LIN {X 0,Y 337.029,Z 979.559,A -85,B 0,C 180,E1 7222.353,E2 7222.353} C_VEL
LIN {X 0,Y 341.956,Z 956.533,A -85,B 0,C 180,E1 7221.821,E2 7221.821} C_VEL
LIN {X 0,Y 345.106,Z 934.145,A -85,B 0,C 180,E1 7221.412,E2 7221.412} C_VEL
LIN {X 0,Y 361.472,Z 765.013,A -85,B 0,C 180,E1 7218.829,E2 7218.829} C_VEL
LIN {X 0,Y 358.291,Z 755.839,A -85,B 0,C 180,E1 7216.122,E2 7216.122} C_VEL
LIN {X 0,Y 355.543,Z 748.18,A -85,B 0,C 180,E1 7213.167,E2 7213.167} C_VEL
LIN {X 0,Y 353.615,Z 742.614,A -85,B 0,C 180,E1 7210.344,E2 7210.344} C_VEL
LIN {X 0,Y 352.385,Z 739.021,A -85,B 0,C 180,E1 7207.664,E2 7207.664} C_VEL
LIN {X 0,Y 351.824,Z 736.43,A -85,B 0,C 180,E1 7205.055,E2 7205.055} C_VEL
LIN {X 0,Y 352.166,Z 735.346,A -85,B 0,C 180,E1 7200.651,E2 7200.651} C_VEL
LIN {X 0,Y 353.212,Z 736.345,A -85,B 0,C 180,E1 7197.891,E2 7197.891} C_VEL
LIN {X 0,Y 354.815,Z 738.293,A -85,B 0,C 180,E1 7195.312,E2 7195.312} C_VEL
LIN {X 0,Y 357.247,Z 742.275,A -85,B 0,C 180,E1 7192.441,E2 7192.441} C_VEL
LIN {X 0,Y 359.812,Z 746.722,A -85,B 0,C 180,E1 7190.079,E2 7190.079} C_VEL
LIN {X 0,Y 363.341,Z 753.377,A -85,B 0,C 180,E1 7187.385,E2 7187.385} C_VEL
LIN {X 0,Y 361.606,Z 770.162,A -85,B 0,C 180,E1 7187.124,E2 7187.124} C_VEL
LIN {X 0,Y 360.533,Z 777.852,A -85,B 0,C 180,E1 7187.159,E2 7187.159} C_VEL
LIN {X 0,Y 356.723,Z 798.361,A -85,B 0,C 180,E1 7187.805,E2 7187.805} C_VEL
LIN {X 0,Y 355.838,Z 804.96,A -85,B 0,C 180,E1 7187.82,E2 7187.82} C_VEL
LIN {X 0,Y 342.283,Z 933.926,A -85,B 0,C 180,E1 7185.77,E2 7185.77} C_VEL
LIN {X 0,Y 338.154,Z 957.934,A -85,B 0,C 180,E1 7185.264,E2 7185.264} C_VEL
LIN {X 0,Y 333.158,Z 979.434,A -85,B 0,C 180,E1 7184.668,E2 7184.668} C_VEL
LIN {X 0,Y 326.772,Z 1000.882,A -85,B 0,C 180,E1 7183.899,E2 7183.899} C_VEL
LIN {X 0,Y 319.517,Z 1021.265,A -85,B 0,C 180,E1 7182.976,E2 7182.976} C_VEL
LIN {X 0,Y 310.546,Z 1042.479,A -85,B 0,C 180,E1 7181.769,E2 7181.769} C_VEL
LIN {X 0,Y 300.999,Z 1062.082,A -85,B 0,C 180,E1 7180.396,E2 7180.396} C_VEL
LIN {X 0,Y 289.845,Z 1081.992,A -85,B 0,C 180,E1 7178.654,E2 7178.654} C_VEL
LIN {X 0,Y 278.251,Z 1100.526,A -85,B 0,C 180,E1 7176.65,E2 7176.65} C_VEL
LIN {X 0,Y 266.028,Z 1117.83,A -85,B 0,C 180,E1 7174.289,E2 7174.289} C_VEL
LIN {X 0,Y 253.22,Z 1134.476,A -85,B 0,C 180,E1 7171.459,E2 7171.459} C_VEL
LIN {X 0,Y 240.898,Z 1149.035,A -85,B 0,C 180,E1 7168.305,E2 7168.305} C_VEL
LIN {X 0,Y 227.747,Z 1163.57,A -85,B 0,C 180,E1 7164.31,E2 7164.31} C_VEL
LIN {X 0,Y 216.336,Z 1175.4,A -85,B 0,C 180,E1 7160.104,E2 7160.104} C_VEL
LIN {X 0,Y 204.152,Z 1187.573,A -85,B 0,C 180,E1 7154.456,E2 7154.456} C_VEL
LIN {X 0,Y 194.783,Z 1196.854,A -85,B 0,C 180,E1 7148.774,E2 7148.774} C_VEL
LIN {X 0,Y 186.937,Z 1204.75,A -85,B 0,C 180,E1 7142.316,E2 7142.316} C_VEL
LIN {X 0,Y 181.505,Z 1210.761,A -85,B 0,C 180,E1 7135.797,E2 7135.797} C_VEL
LIN {X 0,Y 177.788,Z 1215.641,A -85,B 0,C 180,E1 7128.357,E2 7128.357} C_VEL
LIN {X 0,Y 176.331,Z 1218.412,A -85,B 0,C 180,E1 7122.111,E2 7122.111} C_VEL
LIN {X 0,Y 175.975,Z 1220.093,A -85,B 0,C 180,E1 7115.87,E2 7115.87} C_VEL
LIN {X 0,Y 176.025,Z 1220.645,A -85,B 0,C 180,E1 7110,E2 7110} C_VEL
LIN {X 0,Y 175.975,Z 1220.076,A -85,B 0,C 180,E1 7104.13,E2 7104.13} C_VEL
LIN {X 0,Y 176.331,Z 1218.382,A -85,B 0,C 180,E1 7097.889,E2 7097.889} C_VEL
LIN {X 0,Y 177.901,Z 1215.431,A -85,B 0,C 180,E1 7091.315,E2 7091.315} C_VEL
LIN {X 0,Y 181.934,Z 1210.166,A -85,B 0,C 180,E1 7083.567,E2 7083.567} C_VEL
LIN {X 0,Y 187.569,Z 1204.025,A -85,B 0,C 180,E1 7077.063,E2 7077.063} C_VEL
LIN {X 0,Y 195.996,Z 1195.489,A -85,B 0,C 180,E1 7070.381,E2 7070.381} C_VEL
LIN {X 0,Y 205.627,Z 1186.035,A -85,B 0,C 180,E1 7064.772,E2 7064.772} C_VEL
LIN {X 0,Y 216.893,Z 1174.659,A -85,B 0,C 180,E1 7059.659,E2 7059.659} C_VEL
LIN {X 0,Y 229.005,Z 1162.095,A -85,B 0,C 180,E1 7055.268,E2 7055.268} C_VEL
LIN {X 0,Y 241.566,Z 1148.034,A -85,B 0,C 180,E1 7051.499,E2 7051.499} C_VEL
LIN {X 0,Y 254.307,Z 1132.865,A -85,B 0,C 180,E1 7048.273,E2 7048.273} C_VEL
LIN {X 0,Y 266.218,Z 1117.253,A -85,B 0,C 180,E1 7045.659,E2 7045.659} C_VEL
LIN {X 0,Y 278.624,Z 1099.559,A -85,B 0,C 180,E1 7043.268,E2 7043.268} C_VEL
LIN {X 0,Y 289.825,Z 1081.596,A -85,B 0,C 180,E1 7041.336,E2 7041.336} C_VEL
LIN {X 0,Y 300.817,Z 1061.918,A -85,B 0,C 180,E1 7039.616,E2 7039.616} C_VEL
LIN {X 0,Y 310.102,Z 1042.861,A -85,B 0,C 180,E1 7038.277,E2 7038.277} C_VEL
LIN {X 0,Y 319.595,Z 1020.331,A -85,B 0,C 180,E1 7036.999,E2 7036.999} C_VEL
LIN {X 0,Y 327.182,Z 998.816,A -85,B 0,C 180,E1 7036.034,E2 7036.034} C_VEL
LIN {X 0,Y 333.952,Z 975.076,A -85,B 0,C 180,E1 7035.212,E2 7035.212} C_VEL
LIN {X 0,Y 339.074,Z 952.161,A -85,B 0,C 180,E1 7034.611,E2 7034.611} C_VEL
LIN {X 0,Y 342.693,Z 928.355,A -85,B 0,C 180,E1 7034.15,E2 7034.15} C_VEL
LIN {X 0,Y 360.379,Z 758.499,A -85,B 0,C 180,E1 7031.465,E2 7031.465} C_VEL
LIN {X 0,Y 356.925,Z 751.817,A -85,B 0,C 180,E1 7028.539,E2 7028.539} C_VEL
LIN {X 0,Y 354.566,Z 747.889,A -85,B 0,C 180,E1 7026.07,E2 7026.07} C_VEL
LIN {X 0,Y 352.955,Z 745.226,A -85,B 0,C 180,E1 7023.899,E2 7023.899} C_VEL
LIN {X 0,Y 351.105,Z 743.014,A -85,B 0,C 180,E1 7020.163,E2 7020.163} C_VEL
LIN {X 0,Y 350.436,Z 743.287,A -85,B 0,C 180,E1 7016.892,E2 7016.892} C_VEL
LIN {X 0,Y 350.601,Z 744.712,A -85,B 0,C 180,E1 7014.107,E2 7014.107} C_VEL
LIN {X 0,Y 351.499,Z 748.289,A -85,B 0,C 180,E1 7011.081,E2 7011.081} C_VEL
LIN {X 0,Y 352.83,Z 752.197,A -85,B 0,C 180,E1 7008.641,E2 7008.641} C_VEL
LIN {X 0,Y 355.185,Z 759.277,A -85,B 0,C 180,E1 7005.565,E2 7005.565} C_VEL
LIN {X 0,Y 357.437,Z 765.972,A -85,B 0,C 180,E1 7003.296,E2 7003.296} C_VEL
LIN {X 0,Y 358.652,Z 769.729,A -85,B 0,C 180,E1 7002.216,E2 7002.216} C_VEL
LIN {X 0,Y 341.49,Z 941.423,A -85,B 0,C 180,E1 6999.633,E2 6999.633} C_VEL
LIN {X 0,Y 337.472,Z 964.923,A -85,B 0,C 180,E1 6999.174,E2 6999.174} C_VEL
LIN {X 0,Y 332.156,Z 987.28,A -85,B 0,C 180,E1 6998.628,E2 6998.628} C_VEL
LIN {X 0,Y 325.487,Z 1008.737,A -85,B 0,C 180,E1 6997.92,E2 6997.92} C_VEL
LIN {X 0,Y 317.241,Z 1030.712,A -85,B 0,C 180,E1 6996.971,E2 6996.971} C_VEL
LIN {X 0,Y 308.826,Z 1049.617,A -85,B 0,C 180,E1 6995.924,E2 6995.924} C_VEL
LIN {X 0,Y 298.079,Z 1070.431,A -85,B 0,C 180,E1 6994.464,E2 6994.464} C_VEL
LIN {X 0,Y 287.177,Z 1088.966,A -85,B 0,C 180,E1 6992.819,E2 6992.819} C_VEL
LIN {X 0,Y 275.368,Z 1106.536,A -85,B 0,C 180,E1 6990.838,E2 6990.838} C_VEL
LIN {X 0,Y 263.584,Z 1122.475,A -85,B 0,C 180,E1 6988.594,E2 6988.594} C_VEL
LIN {X 0,Y 250.684,Z 1138.039,A -85,B 0,C 180,E1 6985.778,E2 6985.778} C_VEL
LIN {X 0,Y 237.366,Z 1152.752,A -85,B 0,C 180,E1 6982.352,E2 6982.352} C_VEL
LIN {X 0,Y 225.05,Z 1165.313,A -85,B 0,C 180,E1 6978.547,E2 6978.547} C_VEL
LIN {X 0,Y 213.031,Z 1176.669,A -85,B 0,C 180,E1 6973.998,E2 6973.998} C_VEL
LIN {X 0,Y 202.334,Z 1186.397,A -85,B 0,C 180,E1 6968.872,E2 6968.872} C_VEL
LIN {X 0,Y 193.318,Z 1194.256,A -85,B 0,C 180,E1 6963.246,E2 6963.246} C_VEL
LIN {X 0,Y 185.318,Z 1201.367,A -85,B 0,C 180,E1 6956.258,E2 6956.258} C_VEL
LIN {X 0,Y 180.263,Z 1206.2,A -85,B 0,C 180,E1 6949.439,E2 6949.439} C_VEL
LIN {X 0,Y 177.256,Z 1209.525,A -85,B 0,C 180,E1 6942.047,E2 6942.047} C_VEL
LIN {X 0,Y 176.192,Z 1211.235,A -85,B 0,C 180,E1 6935.209,E2 6935.209} C_VEL
LIN {X 0,Y 176.053,Z 1211.594,A -85,B 0,C 180,E1 6929.024,E2 6929.024} C_VEL
LIN {X 0,Y 176.351,Z 1210.882,A -85,B 0,C 180,E1 6922.835,E2 6922.835} C_VEL
LIN {X 0,Y 177.913,Z 1208.822,A -85,B 0,C 180,E1 6915.684,E2 6915.684} C_VEL
LIN {X 0,Y 181.579,Z 1204.916,A -85,B 0,C 180,E1 6908.35,E2 6908.35} C_VEL
LIN {X 0,Y 187.946,Z 1199.095,A -85,B 0,C 180,E1 6901.046,E2 6901.046} C_VEL
LIN {X 0,Y 195.617,Z 1192.379,A -85,B 0,C 180,E1 6895.078,E2 6895.078} C_VEL
LIN {X 0,Y 205.605,Z 1183.544,A -85,B 0,C 180,E1 6889.335,E2 6889.335} C_VEL
LIN {X 0,Y 216.822,Z 1173.386,A -85,B 0,C 180,E1 6884.376,E2 6884.376} C_VEL
LIN {X 0,Y 228.831,Z 1161.702,A -85,B 0,C 180,E1 6880.125,E2 6880.125} C_VEL
LIN {X 0,Y 241.968,Z 1148.06,A -85,B 0,C 180,E1 6876.315,E2 6876.315} C_VEL
LIN {X 0,Y 253.902,Z 1134.56,A -85,B 0,C 180,E1 6873.4,E2 6873.4} C_VEL
LIN {X 0,Y 267.191,Z 1118.005,A -85,B 0,C 180,E1 6870.607,E2 6870.607} C_VEL
LIN {X 0,Y 279.516,Z 1101.047,A -85,B 0,C 180,E1 6868.362,E2 6868.362} C_VEL
LIN {X 0,Y 291.037,Z 1083.022,A -85,B 0,C 180,E1 6866.498,E2 6866.498} C_VEL
LIN {X 0,Y 302.045,Z 1063.664,A -85,B 0,C 180,E1 6864.904,E2 6864.904} C_VEL
LIN {X 0,Y 311.514,Z 1044.454,A -85,B 0,C 180,E1 6863.655,E2 6863.655} C_VEL
LIN {X 0,Y 320.499,Z 1023.203,A -85,B 0,C 180,E1 6862.565,E2 6862.565} C_VEL
LIN {X 0,Y 327.791,Z 1002.724,A -85,B 0,C 180,E1 6861.75,E2 6861.75} C_VEL
LIN {X 0,Y 334.252,Z 980.148,A -85,B 0,C 180,E1 6861.076,E2 6861.076} C_VEL
LIN {X 0,Y 339.282,Z 957.394,A -85,B 0,C 180,E1 6860.559,E2 6860.559} C_VEL
LIN {X 0,Y 342.592,Z 934.57,A -85,B 0,C 180,E1 6860.148,E2 6860.148} C_VEL
LIN {X 0,Y 358.93,Z 769.805,A -85,B 0,C 180,E1 6857.677,E2 6857.677} C_VEL
LIN {X 0,Y 355.989,Z 761.006,A -85,B 0,C 180,E1 6854.892,E2 6854.892} C_VEL
LIN {X 0,Y 353.97,Z 755.084,A -85,B 0,C 180,E1 6852.48,E2 6852.48} C_VEL
LIN {X 0,Y 352.395,Z 750.208,A -85,B 0,C 180,E1 6849.967,E2 6849.967} C_VEL
LIN {X 0,Y 351.295,Z 746.748,A -85,B 0,C 180,E1 6847.359,E2 6847.359} C_VEL
LIN {X 0,Y 350.827,Z 744.326,A -85,B 0,C 180,E1 6844.905,E2 6844.905} C_VEL
LIN {X 0,Y 351.177,Z 743.286,A -85,B 0,C 180,E1 6840.653,E2 6840.653} C_VEL
LIN {X 0,Y 352.164,Z 744.248,A -85,B 0,C 180,E1 6837.999,E2 6837.999} C_VEL
LIN {X 0,Y 353.698,Z 746.195,A -85,B 0,C 180,E1 6835.46,E2 6835.46} C_VEL
LIN {X 0,Y 356.004,Z 750.089,A -85,B 0,C 180,E1 6832.658,E2 6832.658} C_VEL
LIN {X 0,Y 358.693,Z 754.882,A -85,B 0,C 180,E1 6830.129,E2 6830.129} C_VEL
LIN {X 0,Y 360.649,Z 758.948,A -85,B 0,C 180,E1 6828.524,E2 6828.524} C_VEL
LIN {X 0,Y 355.838,Z 804.96,A -85,B 0,C 180,E1 6827.82,E2 6827.82} C_VEL
LIN {X 0,Y 354.777,Z 812.65,A -85,B 0,C 180,E1 6827.857,E2 6827.857} C_VEL
LIN {X 0,Y 351.023,Z 833.156,A -85,B 0,C 180,E1 6828.524,E2 6828.524} C_VEL
LIN {X 0,Y 350.133,Z 839.755,A -85,B 0,C 180,E1 6828.543,E2 6828.543} C_VEL
LIN {X 0,Y 339.9,Z 934.846,A -85,B 0,C 180,E1 6827.045,E2 6827.045} C_VEL
LIN {X 0,Y 335.705,Z 958.6,A -85,B 0,C 180,E1 6826.554,E2 6826.554} C_VEL
LIN {X 0,Y 330.459,Z 980.726,A -85,B 0,C 180,E1 6825.954,E2 6825.954} C_VEL
LIN {X 0,Y 323.727,Z 1002.609,A -85,B 0,C 180,E1 6825.178,E2 6825.178} C_VEL
LIN {X 0,Y 315.704,Z 1024.466,A -85,B 0,C 180,E1 6824.194,E2 6824.194} C_VEL
LIN {X 0,Y 306.366,Z 1045.56,A -85,B 0,C 180,E1 6822.986,E2 6822.986} C_VEL
LIN {X 0,Y 295.733,Z 1066.415,A -85,B 0,C 180,E1 6821.506,E2 6821.506} C_VEL
LIN {X 0,Y 285.197,Z 1084.461,A -85,B 0,C 180,E1 6819.905,E2 6819.905} C_VEL
LIN {X 0,Y 272.268,Z 1104.152,A -85,B 0,C 180,E1 6817.733,E2 6817.733} C_VEL
LIN {X 0,Y 260.434,Z 1120.317,A -85,B 0,C 180,E1 6815.49,E2 6815.49} C_VEL
LIN {X 0,Y 246.783,Z 1137.196,A -85,B 0,C 180,E1 6812.535,E2 6812.535} C_VEL
LIN {X 0,Y 233.842,Z 1151.914,A -85,B 0,C 180,E1 6809.253,E2 6809.253} C_VEL
LIN {X 0,Y 220.408,Z 1165.925,A -85,B 0,C 180,E1 6805.194,E2 6805.194} C_VEL
LIN {X 0,Y 208.173,Z 1178.082,A -85,B 0,C 180,E1 6800.649,E2 6800.649} C_VEL
LIN {X 0,Y 196.781,Z 1188.765,A -85,B 0,C 180,E1 6795.345,E2 6795.345} C_VEL
LIN {X 0,Y 186.709,Z 1198.208,A -85,B 0,C 180,E1 6789.191,E2 6789.191} C_VEL
LIN {X 0,Y 178.738,Z 1205.78,A -85,B 0,C 180,E1 6782.481,E2 6782.481} C_VEL
LIN {X 0,Y 172.554,Z 1212.286,A -85,B 0,C 180,E1 6774.527,E2 6774.527} C_VEL
LIN {X 0,Y 169.474,Z 1216.272,A -85,B 0,C 180,E1 6767.511,E2 6767.511} C_VEL
LIN {X 0,Y 168.095,Z 1219.159,A -85,B 0,C 180,E1 6759.587,E2 6759.587} C_VEL
LIN {X 0,Y 167.988,Z 1220.21,A -85,B 0,C 180,E1 6753.412,E2 6753.412} C_VEL
LIN {X 0,Y 168.009,Z 1220.326,A -85,B 0,C 180,E1 6748.295,E2 6748.295} C_VEL
LIN {X 0,Y 167.997,Z 1219.652,A -85,B 0,C 180,E1 6742.82,E2 6742.82} C_VEL
LIN {X 0,Y 168.51,Z 1217.933,A -85,B 0,C 180,E1 6736.62,E2 6736.62} C_VEL
LIN {X 0,Y 170.726,Z 1214.534,A -85,B 0,C 180,E1 6729.069,E2 6729.069} C_VEL
LIN {X 0,Y 175.265,Z 1209.229,A -85,B 0,C 180,E1 6721.471,E2 6721.471} C_VEL
LIN {X 0,Y 182.19,Z 1202.401,A -85,B 0,C 180,E1 6714.317,E2 6714.317} C_VEL
LIN {X 0,Y 191.024,Z 1194.007,A -85,B 0,C 180,E1 6707.935,E2 6707.935} C_VEL
LIN {X 0,Y 201.99,Z 1183.772,A -85,B 0,C 180,E1 6702.055,E2 6702.055} C_VEL
LIN {X 0,Y 212.898,Z 1173.24,A -85,B 0,C 180,E1 6697.468,E2 6697.468} C_VEL
LIN {X 0,Y 226.306,Z 1159.694,A -85,B 0,C 180,E1 6692.918,E2 6692.918} C_VEL
LIN {X 0,Y 238.766,Z 1146.183,A -85,B 0,C 180,E1 6689.423,E2 6689.423} C_VEL
LIN {X 0,Y 252.747,Z 1129.72,A -85,B 0,C 180,E1 6686.104,E2 6686.104} C_VEL
LIN {X 0,Y 265.241,Z 1113.644,A -85,B 0,C 180,E1 6683.553,E2 6683.553} C_VEL
LIN {X 0,Y 277.898,Z 1095.46,A -85,B 0,C 180,E1 6681.273,E2 6681.273} C_VEL
LIN {X 0,Y 289.428,Z 1077.105,A -85,B 0,C 180,E1 6679.421,E2 6679.421} C_VEL
LIN {X 0,Y 300.367,Z 1057.12,A -85,B 0,C 180,E1 6677.819,E2 6677.819} C_VEL
LIN {X 0,Y 310.441,Z 1036.194,A -85,B 0,C 180,E1 6676.465,E2 6676.465} C_VEL
LIN {X 0,Y 318.459,Z 1016.545,A -85,B 0,C 180,E1 6675.447,E2 6675.447} C_VEL
LIN {X 0,Y 326.104,Z 994.574,A -85,B 0,C 180,E1 6674.527,E2 6674.527} C_VEL
LIN {X 0,Y 332.333,Z 972.111,A -85,B 0,C 180,E1 6673.804,E2 6673.804} C_VEL
LIN {X 0,Y 337.707,Z 946.629,A -85,B 0,C 180,E1 6673.192,E2 6673.192} C_VEL
LIN {X 0,Y 341.067,Z 923.287,A -85,B 0,C 180,E1 6672.775,E2 6672.775} C_VEL
LIN {X 0,Y 357.834,Z 764.018,A -85,B 0,C 180,E1 6670.302,E2 6670.302} C_VEL
LIN {X 0,Y 354.927,Z 758.432,A -85,B 0,C 180,E1 6667.609,E2 6667.609} C_VEL
LIN {X 0,Y 353.161,Z 755.368,A -85,B 0,C 180,E1 6665.606,E2 6665.606} C_VEL
LIN {X 0,Y 351.853,Z 753.098,A -85,B 0,C 180,E1 6663.748,E2 6663.748} C_VEL
LIN {X 0,Y 350.116,Z 750.958,A -85,B 0,C 180,E1 6660.164,E2 6660.164} C_VEL
LIN {X 0,Y 349.463,Z 751.211,A -85,B 0,C 180,E1 6656.982,E2 6656.982} C_VEL
LIN {X 0,Y 349.579,Z 752.427,A -85,B 0,C 180,E1 6654.419,E2 6654.419} C_VEL
LIN {X 0,Y 350.452,Z 756.238,A -85,B 0,C 180,E1 6651.22,E2 6651.22} C_VEL
LIN {X 0,Y 351.633,Z 759.943,A -85,B 0,C 180,E1 6648.934,E2 6648.934} C_VEL
LIN {X 0,Y 353.806,Z 766.851,A -85,B 0,C 180,E1 6645.934,E2 6645.934} C_VEL
LIN {X 0,Y 355.94,Z 773.524,A -85,B 0,C 180,E1 6643.685,E2 6643.685} C_VEL
LIN {X 0,Y 356.225,Z 774.674,A -85,B 0,C 180,E1 6643.392,E2 6643.392} C_VEL
LIN {X 0,Y 339.205,Z 941.139,A -85,B 0,C 180,E1 6640.929,E2 6640.929} C_VEL
LIN {X 0,Y 335.127,Z 964.63,A -85,B 0,C 180,E1 6640.482,E2 6640.482} C_VEL
LIN {X 0,Y 329.687,Z 987.161,A -85,B 0,C 180,E1 6639.95,E2 6639.95} C_VEL
LIN {X 0,Y 323.312,Z 1007.456,A -85,B 0,C 180,E1 6639.308,E2 6639.308} C_VEL
LIN {X 0,Y 315.069,Z 1029.359,A -85,B 0,C 180,E1 6638.407,E2 6638.407} C_VEL
LIN {X 0,Y 306.079,Z 1049.291,A -85,B 0,C 180,E1 6637.343,E2 6637.343} C_VEL
LIN {X 0,Y 295.167,Z 1070.096,A -85,B 0,C 180,E1 6635.93,E2 6635.93} C_VEL
LIN {X 0,Y 284.01,Z 1088.714,A -85,B 0,C 180,E1 6634.322,E2 6634.322} C_VEL
LIN {X 0,Y 271.939,Z 1106.33,A -85,B 0,C 180,E1 6632.387,E2 6632.387} C_VEL
LIN {X 0,Y 259.478,Z 1122.768,A -85,B 0,C 180,E1 6630.112,E2 6630.112} C_VEL
LIN {X 0,Y 246.74,Z 1137.745,A -85,B 0,C 180,E1 6627.445,E2 6627.445} C_VEL
LIN {X 0,Y 233.226,Z 1152.292,A -85,B 0,C 180,E1 6624.121,E2 6624.121} C_VEL
LIN {X 0,Y 221.236,Z 1164.119,A -85,B 0,C 180,E1 6620.608,E2 6620.608} C_VEL
LIN {X 0,Y 208.421,Z 1175.889,A -85,B 0,C 180,E1 6616.021,E2 6616.021} C_VEL
LIN {X 0,Y 197.073,Z 1185.776,A -85,B 0,C 180,E1 6610.881,E2 6610.881} C_VEL
LIN {X 0,Y 186.99,Z 1194.129,A -85,B 0,C 180,E1 6604.9,E2 6604.9} C_VEL
LIN {X 0,Y 178.69,Z 1201.085,A -85,B 0,C 180,E1 6598.036,E2 6598.036} C_VEL
LIN {X 0,Y 173.051,Z 1206.011,A -85,B 0,C 180,E1 6590.991,E2 6590.991} C_VEL
LIN {X 0,Y 169.48,Z 1209.623,A -85,B 0,C 180,E1 6582.955,E2 6582.955} C_VEL
LIN {X 0,Y 168.261,Z 1211.31,A -85,B 0,C 180,E1 6576.14,E2 6576.14} C_VEL
LIN {X 0,Y 168.054,Z 1211.842,A -85,B 0,C 180,E1 6569.659,E2 6569.659} C_VEL
LIN {X 0,Y 168.315,Z 1211.216,A -85,B 0,C 180,E1 6563.177,E2 6563.177} C_VEL
LIN {X 0,Y 169.652,Z 1209.467,A -85,B 0,C 180,E1 6556.365,E2 6556.365} C_VEL
LIN {X 0,Y 173.416,Z 1205.721,A -85,B 0,C 180,E1 6548.346,E2 6548.346} C_VEL
LIN {X 0,Y 179.567,Z 1200.472,A -85,B 0,C 180,E1 6541.025,E2 6541.025} C_VEL
LIN {X 0,Y 187.732,Z 1193.622,A -85,B 0,C 180,E1 6534.512,E2 6534.512} C_VEL
LIN {X 0,Y 197.975,Z 1185.108,A -85,B 0,C 180,E1 6528.578,E2 6528.578} C_VEL
LIN {X 0,Y 208.881,Z 1175.638,A -85,B 0,C 180,E1 6523.714,E2 6523.714} C_VEL
LIN {X 0,Y 221.785,Z 1163.78,A -85,B 0,C 180,E1 6519.137,E2 6519.137} C_VEL
LIN {X 0,Y 234.717,Z 1151.027,A -85,B 0,C 180,E1 6515.406,E2 6515.406} C_VEL
LIN {X 0,Y 248.074,Z 1136.498,A -85,B 0,C 180,E1 6512.178,E2 6512.178} C_VEL
LIN {X 0,Y 261.258,Z 1120.816,A -85,B 0,C 180,E1 6509.464,E2 6509.464} C_VEL
LIN {X 0,Y 273.392,Z 1104.677,A -85,B 0,C 180,E1 6507.289,E2 6507.289} C_VEL
LIN {X 0,Y 286.32,Z 1085.401,A -85,B 0,C 180,E1 6505.251,E2 6505.251} C_VEL
LIN {X 0,Y 297.51,Z 1066.502,A -85,B 0,C 180,E1 6503.68,E2 6503.68} C_VEL
LIN {X 0,Y 307.645,Z 1046.583,A -85,B 0,C 180,E1 6502.387,E2 6502.387} C_VEL
LIN {X 0,Y 316.66,Z 1026.189,A -85,B 0,C 180,E1 6501.336,E2 6501.336} C_VEL
LIN {X 0,Y 324.05,Z 1006.131,A -85,B 0,C 180,E1 6500.537,E2 6500.537} C_VEL
LIN {X 0,Y 330.956,Z 983.433,A -85,B 0,C 180,E1 6499.847,E2 6499.847} C_VEL
LIN {X 0,Y 336.032,Z 961.712,A -85,B 0,C 180,E1 6499.351,E2 6499.351} C_VEL
LIN {X 0,Y 339.923,Z 937.638,A -85,B 0,C 180,E1 6498.909,E2 6498.909} C_VEL
LIN {X 0,Y 356.513,Z 774.64,A -85,B 0,C 180,E1 6496.497,E2 6496.497} C_VEL
LIN {X 0,Y 354.177,Z 767.326,A -85,B 0,C 180,E1 6494.051,E2 6494.051} C_VEL
LIN {X 0,Y 352.392,Z 761.804,A -85,B 0,C 180,E1 6491.705,E2 6491.705} C_VEL
LIN {X 0,Y 351.108,Z 757.576,A -85,B 0,C 180,E1 6489.425,E2 6489.425} C_VEL
LIN {X 0,Y 350.214,Z 754.474,A -85,B 0,C 180,E1 6487.052,E2 6487.052} C_VEL
LIN {X 0,Y 349.833,Z 752.223,A -85,B 0,C 180,E1 6484.755,E2 6484.755} C_VEL
LIN {X 0,Y 350.188,Z 751.226,A -85,B 0,C 180,E1 6480.654,E2 6480.654} C_VEL
LIN {X 0,Y 351.159,Z 752.206,A -85,B 0,C 180,E1 6478.019,E2 6478.019} C_VEL
LIN {X 0,Y 352.583,Z 754.095,A -85,B 0,C 180,E1 6475.609,E2 6475.609} C_VEL
LIN {X 0,Y 354.688,Z 757.761,A -85,B 0,C 180,E1 6472.956,E2 6472.956} C_VEL
LIN {X 0,Y 357.293,Z 762.562,A -85,B 0,C 180,E1 6470.415,E2 6470.415} C_VEL
LIN {X 0,Y 358.11,Z 764.564,A -85,B 0,C 180,E1 6469.679,E2 6469.679} C_VEL
LIN {X 0,Y 350.133,Z 839.755,A -85,B 0,C 180,E1 6468.543,E2 6468.543} C_VEL
LIN {X 0,Y 349.068,Z 847.445,A -85,B 0,C 180,E1 6468.585,E2 6468.585} C_VEL
LIN {X 0,Y 345.369,Z 867.952,A -85,B 0,C 180,E1 6469.273,E2 6469.273} C_VEL
LIN {X 0,Y 344.489,Z 874.551,A -85,B 0,C 180,E1 6469.291,E2 6469.291} C_VEL
LIN {X 0,Y 337.551,Z 936.843,A -85,B 0,C 180,E1 6468.32,E2 6468.32} C_VEL
LIN {X 0,Y 333.239,Z 960.153,A -85,B 0,C 180,E1 6467.842,E2 6467.842} C_VEL
LIN {X 0,Y 327.792,Z 982.422,A -85,B 0,C 180,E1 6467.245,E2 6467.245} C_VEL
LIN {X 0,Y 321.246,Z 1003.171,A -85,B 0,C 180,E1 6466.527,E2 6466.527} C_VEL
LIN {X 0,Y 313.137,Z 1024.834,A -85,B 0,C 180,E1 6465.578,E2 6465.578} C_VEL
LIN {X 0,Y 303.637,Z 1045.904,A -85,B 0,C 180,E1 6464.404,E2 6464.404} C_VEL
LIN {X 0,Y 292.807,Z 1066.708,A -85,B 0,C 180,E1 6462.965,E2 6462.965} C_VEL
LIN {X 0,Y 281.943,Z 1084.92,A -85,B 0,C 180,E1 6461.387,E2 6461.387} C_VEL
LIN {X 0,Y 268.435,Z 1104.934,A -85,B 0,C 180,E1 6459.214,E2 6459.214} C_VEL
LIN {X 0,Y 255.929,Z 1121.54,A -85,B 0,C 180,E1 6456.932,E2 6456.932} C_VEL
LIN {X 0,Y 242.028,Z 1138.102,A -85,B 0,C 180,E1 6454.029,E2 6454.029} C_VEL
LIN {X 0,Y 228.278,Z 1153.184,A -85,B 0,C 180,E1 6450.647,E2 6450.647} C_VEL
LIN {X 0,Y 214.757,Z 1166.676,A -85,B 0,C 180,E1 6446.674,E2 6446.674} C_VEL
LIN {X 0,Y 201.199,Z 1179.44,A -85,B 0,C 180,E1 6441.737,E2 6441.737} C_VEL
LIN {X 0,Y 189.982,Z 1189.481,A -85,B 0,C 180,E1 6436.575,E2 6436.575} C_VEL
LIN {X 0,Y 179.06,Z 1199.089,A -85,B 0,C 180,E1 6429.952,E2 6429.952} C_VEL
LIN {X 0,Y 171.157,Z 1206.193,A -85,B 0,C 180,E1 6423.307,E2 6423.307} C_VEL
LIN {X 0,Y 164.757,Z 1212.431,A -85,B 0,C 180,E1 6415.138,E2 6415.138} C_VEL
LIN {X 0,Y 161.476,Z 1216.4,A -85,B 0,C 180,E1 6407.662,E2 6407.662} C_VEL
LIN {X 0,Y 160.079,Z 1219.099,A -85,B 0,C 180,E1 6399.346,E2 6399.346} C_VEL
LIN {X 0,Y 159.991,Z 1220.03,A -85,B 0,C 180,E1 6393.224,E2 6393.224} C_VEL
LIN {X 0,Y 160.01,Z 1220.122,A -85,B 0,C 180,E1 6388.21,E2 6388.21} C_VEL
LIN {X 0,Y 159.997,Z 1219.446,A -85,B 0,C 180,E1 6382.459,E2 6382.459} C_VEL
LIN {X 0,Y 160.611,Z 1217.724,A -85,B 0,C 180,E1 6375.949,E2 6375.949} C_VEL
LIN {X 0,Y 163.092,Z 1214.322,A -85,B 0,C 180,E1 6368.04,E2 6368.04} C_VEL
LIN {X 0,Y 167.864,Z 1209.203,A -85,B 0,C 180,E1 6360.371,E2 6360.371} C_VEL
LIN {X 0,Y 175.131,Z 1202.553,A -85,B 0,C 180,E1 6353.065,E2 6353.065} C_VEL
LIN {X 0,Y 184.466,Z 1194.201,A -85,B 0,C 180,E1 6346.499,E2 6346.499} C_VEL
LIN {X 0,Y 195.958,Z 1184.065,A -85,B 0,C 180,E1 6340.513,E2 6340.513} C_VEL
LIN {X 0,Y 207.953,Z 1172.995,A -85,B 0,C 180,E1 6335.653,E2 6335.653} C_VEL
LIN {X 0,Y 221.905,Z 1159.43,A -85,B 0,C 180,E1 6331.119,E2 6331.119} C_VEL
LIN {X 0,Y 234.855,Z 1145.859,A -85,B 0,C 180,E1 6327.65,E2 6327.65} C_VEL
LIN {X 0,Y 249.221,Z 1129.413,A -85,B 0,C 180,E1 6324.397,E2 6324.397} C_VEL
LIN {X 0,Y 262.313,Z 1112.987,A -85,B 0,C 180,E1 6321.852,E2 6321.852} C_VEL
LIN {X 0,Y 275.019,Z 1095.075,A -85,B 0,C 180,E1 6319.675,E2 6319.675} C_VEL
LIN {X 0,Y 287.183,Z 1076.016,A -85,B 0,C 180,E1 6317.816,E2 6317.816} C_VEL
LIN {X 0,Y 297.963,Z 1056.604,A -85,B 0,C 180,E1 6316.319,E2 6316.319} C_VEL
LIN {X 0,Y 308,Z 1036.051,A -85,B 0,C 180,E1 6315.035,E2 6315.035} C_VEL
LIN {X 0,Y 316.384,Z 1015.786,A -85,B 0,C 180,E1 6314.023,E2 6314.023} C_VEL
LIN {X 0,Y 324.402,Z 992.707,A -85,B 0,C 180,E1 6313.104,E2 6313.104} C_VEL
LIN {X 0,Y 330.456,Z 970.947,A -85,B 0,C 180,E1 6312.435,E2 6312.435} C_VEL
LIN {X 0,Y 335.63,Z 946.381,A -85,B 0,C 180,E1 6311.871,E2 6311.871} C_VEL
LIN {X 0,Y 339.057,Z 922.733,A -85,B 0,C 180,E1 6311.462,E2 6311.462} C_VEL
LIN {X 0,Y 355.457,Z 769.686,A -85,B 0,C 180,E1 6309.145,E2 6309.145} C_VEL
LIN {X 0,Y 352.697,Z 764.265,A -85,B 0,C 180,E1 6306.266,E2 6306.266} C_VEL
LIN {X 0,Y 350.648,Z 760.861,A -85,B 0,C 180,E1 6303.433,E2 6303.433} C_VEL
LIN {X 0,Y 349.072,Z 758.864,A -85,B 0,C 180,E1 6300,E2 6300} C_VEL
LIN {X 0,Y 348.467,Z 759.196,A -85,B 0,C 180,E1 6296.875,E2 6296.875} C_VEL
LIN {X 0,Y 348.595,Z 760.49,A -85,B 0,C 180,E1 6294.432,E2 6294.432} C_VEL
LIN {X 0,Y 349.334,Z 763.94,A -85,B 0,C 180,E1 6291.523,E2 6291.523} C_VEL
LIN {X 0,Y 350.389,Z 767.507,A -85,B 0,C 180,E1 6289.31,E2 6289.31} C_VEL
LIN {X 0,Y 352.384,Z 774.234,A -85,B 0,C 180,E1 6286.378,E2 6286.378} C_VEL
LIN {X 0,Y 353.955,Z 779.434,A -85,B 0,C 180,E1 6284.59,E2 6284.59} C_VEL
LIN {X 0,Y 337.093,Z 940.877,A -85,B 0,C 180,E1 6282.242,E2 6282.242} C_VEL
LIN {X 0,Y 332.925,Z 964.495,A -85,B 0,C 180,E1 6281.805,E2 6281.805} C_VEL
LIN {X 0,Y 327.578,Z 986.439,A -85,B 0,C 180,E1 6281.307,E2 6281.307} C_VEL
LIN {X 0,Y 321.029,Z 1007.046,A -85,B 0,C 180,E1 6280.683,E2 6280.683} C_VEL
LIN {X 0,Y 313.099,Z 1028.006,A -85,B 0,C 180,E1 6279.862,E2 6279.862} C_VEL
LIN {X 0,Y 303.955,Z 1048.068,A -85,B 0,C 180,E1 6278.839,E2 6278.839} C_VEL
LIN {X 0,Y 292.81,Z 1069.146,A -85,B 0,C 180,E1 6277.469,E2 6277.469} C_VEL
LIN {X 0,Y 281.873,Z 1087.137,A -85,B 0,C 180,E1 6275.979,E2 6275.979} C_VEL
LIN {X 0,Y 269.119,Z 1105.575,A -85,B 0,C 180,E1 6274.04,E2 6274.04} C_VEL
LIN {X 0,Y 256.345,Z 1122.136,A -85,B 0,C 180,E1 6271.823,E2 6271.823} C_VEL
LIN {X 0,Y 243.247,Z 1137.192,A -85,B 0,C 180,E1 6269.214,E2 6269.214} C_VEL
LIN {X 0,Y 229.296,Z 1151.853,A -85,B 0,C 180,E1 6265.945,E2 6265.945} C_VEL
LIN {X 0,Y 216.853,Z 1163.739,A -85,B 0,C 180,E1 6262.471,E2 6262.471} C_VEL
LIN {X 0,Y 202.873,Z 1176.114,A -85,B 0,C 180,E1 6257.67,E2 6257.67} C_VEL
LIN {X 0,Y 190.755,Z 1186.218,A -85,B 0,C 180,E1 6252.346,E2 6252.346} C_VEL
LIN {X 0,Y 180.39,Z 1194.344,A -85,B 0,C 180,E1 6246.375,E2 6246.375} C_VEL
LIN {X 0,Y 171.573,Z 1201.296,A -85,B 0,C 180,E1 6239.309,E2 6239.309} C_VEL
LIN {X 0,Y 165.517,Z 1206.221,A -85,B 0,C 180,E1 6231.995,E2 6231.995} C_VEL
LIN {X 0,Y 161.63,Z 1209.829,A -85,B 0,C 180,E1 6223.596,E2 6223.596} C_VEL
LIN {X 0,Y 160.287,Z 1211.516,A -85,B 0,C 180,E1 6216.447,E2 6216.447} C_VEL
LIN {X 0,Y 160.057,Z 1212.047,A -85,B 0,C 180,E1 6209.642,E2 6209.642} C_VEL
LIN {X 0,Y 160.348,Z 1211.422,A -85,B 0,C 180,E1 6202.836,E2 6202.836} C_VEL
LIN {X 0,Y 161.823,Z 1209.672,A -85,B 0,C 180,E1 6195.691,E2 6195.691} C_VEL
LIN {X 0,Y 165.915,Z 1205.927,A -85,B 0,C 180,E1 6187.314,E2 6187.314} C_VEL
LIN {X 0,Y 172.512,Z 1200.681,A -85,B 0,C 180,E1 6179.719,E2 6179.719} C_VEL
LIN {X 0,Y 181.181,Z 1193.835,A -85,B 0,C 180,E1 6173.021,E2 6173.021} C_VEL
LIN {X 0,Y 191.963,Z 1185.329,A -85,B 0,C 180,E1 6166.974,E2 6166.974} C_VEL
LIN {X 0,Y 203.359,Z 1175.862,A -85,B 0,C 180,E1 6162.062,E2 6162.062} C_VEL
LIN {X 0,Y 217.4,Z 1163.428,A -85,B 0,C 180,E1 6157.283,E2 6157.283} C_VEL
LIN {X 0,Y 230.601,Z 1150.816,A -85,B 0,C 180,E1 6153.645,E2 6153.645} C_VEL
LIN {X 0,Y 244.074,Z 1136.547,A -85,B 0,C 180,E1 6150.53,E2 6150.53} C_VEL
LIN {X 0,Y 257.786,Z 1120.626,A -85,B 0,C 180,E1 6147.831,E2 6147.831} C_VEL
LIN {X 0,Y 270.208,Z 1104.462,A -85,B 0,C 180,E1 6145.707,E2 6145.707} C_VEL
LIN {X 0,Y 282.993,Z 1085.799,A -85,B 0,C 180,E1 6143.782,E2 6143.782} C_VEL
LIN {X 0,Y 293.96,Z 1067.668,A -85,B 0,C 180,E1 6142.307,E2 6142.307} C_VEL
LIN {X 0,Y 304.26,Z 1048.029,A -85,B 0,C 180,E1 6141.049,E2 6141.049} C_VEL
LIN {X 0,Y 313.41,Z 1027.955,A -85,B 0,C 180,E1 6140.028,E2 6140.028} C_VEL
LIN {X 0,Y 321.345,Z 1006.979,A -85,B 0,C 180,E1 6139.208,E2 6139.208} C_VEL
LIN {X 0,Y 328.248,Z 985.035,A -85,B 0,C 180,E1 6138.552,E2 6138.552} C_VEL
LIN {X 0,Y 333.571,Z 962.86,A -85,B 0,C 180,E1 6138.057,E2 6138.057} C_VEL
LIN {X 0,Y 337.762,Z 937.904,A -85,B 0,C 180,E1 6137.608,E2 6137.608} C_VEL
LIN {X 0,Y 354.237,Z 779.666,A -85,B 0,C 180,E1 6135.311,E2 6135.311} C_VEL
LIN {X 0,Y 352.025,Z 772.167,A -85,B 0,C 180,E1 6132.633,E2 6132.633} C_VEL
LIN {X 0,Y 350.132,Z 765.728,A -85,B 0,C 180,E1 6129.451,E2 6129.451} C_VEL
LIN {X 0,Y 349.194,Z 762.369,A -85,B 0,C 180,E1 6126.907,E2 6126.907} C_VEL
LIN {X 0,Y 348.845,Z 760.121,A -85,B 0,C 180,E1 6124.603,E2 6124.603} C_VEL
LIN {X 0,Y 349.242,Z 759.189,A -85,B 0,C 180,E1 6120.492,E2 6120.492} C_VEL
LIN {X 0,Y 350.233,Z 760.271,A -85,B 0,C 180,E1 6117.873,E2 6117.873} C_VEL
LIN {X 0,Y 351.418,Z 761.884,A -85,B 0,C 180,E1 6115.839,E2 6115.839} C_VEL
LIN {X 0,Y 353.474,Z 765.623,A -85,B 0,C 180,E1 6113.147,E2 6113.147} C_VEL
LIN {X 0,Y 355.731,Z 769.938,A -85,B 0,C 180,E1 6110.857,E2 6110.857} C_VEL
LIN {X 0,Y 344.489,Z 874.551,A -85,B 0,C 180,E1 6109.291,E2 6109.291} C_VEL
LIN {X 0,Y 343.432,Z 882.24,A -85,B 0,C 180,E1 6109.334,E2 6109.334} C_VEL
LIN {X 0,Y 339.777,Z 902.737,A -85,B 0,C 180,E1 6110.051,E2 6110.051} C_VEL
LIN {X 0,Y 338.901,Z 909.337,A -85,B 0,C 180,E1 6110.073,E2 6110.073} C_VEL
LIN {X 0,Y 334.923,Z 941.101,A -85,B 0,C 180,E1 6109.571,E2 6109.571} C_VEL
LIN {X 0,Y 330.648,Z 963.067,A -85,B 0,C 180,E1 6109.119,E2 6109.119} C_VEL
LIN {X 0,Y 324.493,Z 986.623,A -85,B 0,C 180,E1 6108.478,E2 6108.478} C_VEL
LIN {X 0,Y 318.135,Z 1006.073,A -85,B 0,C 180,E1 6107.804,E2 6107.804} C_VEL
LIN {X 0,Y 309.125,Z 1028.895,A -85,B 0,C 180,E1 6106.799,E2 6106.799} C_VEL
LIN {X 0,Y 299.768,Z 1048.984,A -85,B 0,C 180,E1 6105.684,E2 6105.684} C_VEL
LIN {X 0,Y 288.759,Z 1069.237,A -85,B 0,C 180,E1 6104.281,E2 6104.281} C_VEL
LIN {X 0,Y 277.082,Z 1088.213,A -85,B 0,C 180,E1 6102.641,E2 6102.641} C_VEL
LIN {X 0,Y 263.949,Z 1106.847,A -85,B 0,C 180,E1 6100.601,E2 6100.601} C_VEL
LIN {X 0,Y 250.358,Z 1124.218,A -85,B 0,C 180,E1 6098.196,E2 6098.196} C_VEL
LIN {X 0,Y 237.26,Z 1139.212,A -85,B 0,C 180,E1 6095.542,E2 6095.542} C_VEL
LIN {X 0,Y 222.851,Z 1154.362,A -85,B 0,C 180,E1 6092.113,E2 6092.113} C_VEL
LIN {X 0,Y 209.645,Z 1167.055,A -85,B 0,C 180,E1 6088.356,E2 6088.356} C_VEL
LIN {X 0,Y 194.919,Z 1180.268,A -85,B 0,C 180,E1 6083.151,E2 6083.151} C_VEL
LIN {X 0,Y 182.735,Z 1190.671,A -85,B 0,C 180,E1 6077.618,E2 6077.618} C_VEL
LIN {X 0,Y 171.885,Z 1199.599,A -85,B 0,C 180,E1 6071.096,E2 6071.096} C_VEL
LIN {X 0,Y 163.279,Z 1206.918,A -85,B 0,C 180,E1 6063.866,E2 6063.866} C_VEL
LIN {X 0,Y 156.903,Z 1212.653,A -85,B 0,C 180,E1 6055.679,E2 6055.679} C_VEL
LIN {X 0,Y 153.267,Z 1216.822,A -85,B 0,C 180,E1 6047.071,E2 6047.071} C_VEL
LIN {X 0,Y 152.059,Z 1219.04,A -85,B 0,C 180,E1 6039.08,E2 6039.08} C_VEL
LIN {X 0,Y 151.993,Z 1219.85,A -85,B 0,C 180,E1 6033.017,E2 6033.017} C_VEL
LIN {X 0,Y 152.003,Z 1219.893,A -85,B 0,C 180,E1 6027.738,E2 6027.738} C_VEL
LIN {X 0,Y 152.017,Z 1219.167,A -85,B 0,C 180,E1 6021.68,E2 6021.68} C_VEL
LIN {X 0,Y 152.81,Z 1217.394,A -85,B 0,C 180,E1 6014.828,E2 6014.828} C_VEL
LIN {X 0,Y 155.883,Z 1213.677,A -85,B 0,C 180,E1 6006.166,E2 6006.166} C_VEL
LIN {X 0,Y 161.034,Z 1208.723,A -85,B 0,C 180,E1 5998.563,E2 5998.563} C_VEL
LIN {X 0,Y 169.297,Z 1201.693,A -85,B 0,C 180,E1 5990.807,E2 5990.807} C_VEL
LIN {X 0,Y 179.044,Z 1193.558,A -85,B 0,C 180,E1 5984.373,E2 5984.373} C_VEL
LIN {X 0,Y 191.857,Z 1182.769,A -85,B 0,C 180,E1 5978.1,E2 5978.1} C_VEL
LIN {X 0,Y 203.891,Z 1172.166,A -85,B 0,C 180,E1 5973.524,E2 5973.524} C_VEL
LIN {X 0,Y 218.636,Z 1158.267,A -85,B 0,C 180,E1 5968.998,E2 5968.998} C_VEL
LIN {X 0,Y 231.842,Z 1144.851,A -85,B 0,C 180,E1 5965.665,E2 5965.665} C_VEL
LIN {X 0,Y 245.923,Z 1129.107,A -85,B 0,C 180,E1 5962.643,E2 5962.643} C_VEL
LIN {X 0,Y 259.772,Z 1112.139,A -85,B 0,C 180,E1 5960.091,E2 5960.091} C_VEL
LIN {X 0,Y 272.785,Z 1094.073,A -85,B 0,C 180,E1 5957.981,E2 5957.981} C_VEL
LIN {X 0,Y 285.255,Z 1074.732,A -85,B 0,C 180,E1 5956.177,E2 5956.177} C_VEL
LIN {X 0,Y 295.766,Z 1056.09,A -85,B 0,C 180,E1 5954.796,E2 5954.796} C_VEL
LIN {X 0,Y 306.426,Z 1034.371,A -85,B 0,C 180,E1 5953.502,E2 5953.502} C_VEL
LIN {X 0,Y 314.507,Z 1015.027,A -85,B 0,C 180,E1 5952.581,E2 5952.581} C_VEL
LIN {X 0,Y 322.652,Z 991.658,A -85,B 0,C 180,E1 5951.695,E2 5951.695} C_VEL
LIN {X 0,Y 328.771,Z 969.786,A -85,B 0,C 180,E1 5951.053,E2 5951.053} C_VEL
LIN {X 0,Y 333.75,Z 946.053,A -85,B 0,C 180,E1 5950.533,E2 5950.533} C_VEL
LIN {X 0,Y 337.213,Z 922.181,A -85,B 0,C 180,E1 5950.134,E2 5950.134} C_VEL
LIN {X 0,Y 353.156,Z 775.477,A -85,B 0,C 180,E1 5947.934,E2 5947.934} C_VEL
LIN {X 0,Y 350.96,Z 771.249,A -85,B 0,C 180,E1 5945.395,E2 5945.395} C_VEL
LIN {X 0,Y 349.483,Z 768.656,A -85,B 0,C 180,E1 5943.166,E2 5943.166} C_VEL
LIN {X 0,Y 348.081,Z 766.807,A -85,B 0,C 180,E1 5940,E2 5940} C_VEL
LIN {X 0,Y 347.483,Z 767.168,A -85,B 0,C 180,E1 5936.826,E2 5936.826} C_VEL
LIN {X 0,Y 347.579,Z 768.237,A -85,B 0,C 180,E1 5934.718,E2 5934.718} C_VEL
LIN {X 0,Y 348.25,Z 771.763,A -85,B 0,C 180,E1 5931.746,E2 5931.746} C_VEL
LIN {X 0,Y 349.201,Z 775.249,A -85,B 0,C 180,E1 5929.607,E2 5929.607} C_VEL
LIN {X 0,Y 351.015,Z 781.723,A -85,B 0,C 180,E1 5926.785,E2 5926.785} C_VEL
LIN {X 0,Y 351.799,Z 784.586,A -85,B 0,C 180,E1 5925.79,E2 5925.79} C_VEL
LIN {X 0,Y 335.168,Z 940.545,A -85,B 0,C 180,E1 5923.572,E2 5923.572} C_VEL
LIN {X 0,Y 330.958,Z 964.097,A -85,B 0,C 180,E1 5923.15,E2 5923.15} C_VEL
LIN {X 0,Y 325.386,Z 986.602,A -85,B 0,C 180,E1 5922.658,E2 5922.658} C_VEL
LIN {X 0,Y 318.485,Z 1007.911,A -85,B 0,C 180,E1 5922.034,E2 5922.034} C_VEL
LIN {X 0,Y 309.999,Z 1029.648,A -85,B 0,C 180,E1 5921.198,E2 5921.198} C_VEL
LIN {X 0,Y 300.727,Z 1049.524,A -85,B 0,C 180,E1 5920.206,E2 5920.206} C_VEL
LIN {X 0,Y 289.406,Z 1070.32,A -85,B 0,C 180,E1 5918.877,E2 5918.877} C_VEL
LIN {X 0,Y 277.439,Z 1089.521,A -85,B 0,C 180,E1 5917.308,E2 5917.308} C_VEL
LIN {X 0,Y 264.801,Z 1107.106,A -85,B 0,C 180,E1 5915.458,E2 5915.458} C_VEL
LIN {X 0,Y 251.036,Z 1124.269,A -85,B 0,C 180,E1 5913.148,E2 5913.148} C_VEL
LIN {X 0,Y 237.675,Z 1139.138,A -85,B 0,C 180,E1 5910.553,E2 5910.553} C_VEL
LIN {X 0,Y 223.401,Z 1153.485,A -85,B 0,C 180,E1 5907.29,E2 5907.29} C_VEL
LIN {X 0,Y 209.961,Z 1165.857,A -85,B 0,C 180,E1 5903.59,E2 5903.59} C_VEL
LIN {X 0,Y 196.877,Z 1176.845,A -85,B 0,C 180,E1 5899.175,E2 5899.175} C_VEL
LIN {X 0,Y 184.51,Z 1186.684,A -85,B 0,C 180,E1 5893.883,E2 5893.883} C_VEL
LIN {X 0,Y 173.461,Z 1194.901,A -85,B 0,C 180,E1 5887.662,E2 5887.662} C_VEL
LIN {X 0,Y 163.85,Z 1201.997,A -85,B 0,C 180,E1 5880.026,E2 5880.026} C_VEL
LIN {X 0,Y 157.573,Z 1206.829,A -85,B 0,C 180,E1 5872.378,E2 5872.378} C_VEL
LIN {X 0,Y 153.689,Z 1210.145,A -85,B 0,C 180,E1 5863.929,E2 5863.929} C_VEL
LIN {X 0,Y 152.253,Z 1211.851,A -85,B 0,C 180,E1 5856.031,E2 5856.031} C_VEL
LIN {X 0,Y 152.062,Z 1212.207,A -85,B 0,C 180,E1 5848.87,E2 5848.87} C_VEL
LIN {X 0,Y 152.43,Z 1211.561,A -85,B 0,C 180,E1 5842.082,E2 5842.082} C_VEL
LIN {X 0,Y 154.278,Z 1209.661,A -85,B 0,C 180,E1 5834.205,E2 5834.205} C_VEL
LIN {X 0,Y 158.723,Z 1205.936,A -85,B 0,C 180,E1 5825.829,E2 5825.829} C_VEL
LIN {X 0,Y 165.921,Z 1200.611,A -85,B 0,C 180,E1 5817.975,E2 5817.975} C_VEL
LIN {X 0,Y 175.233,Z 1193.704,A -85,B 0,C 180,E1 5811.123,E2 5811.123} C_VEL
LIN {X 0,Y 187.236,Z 1184.653,A -85,B 0,C 180,E1 5804.746,E2 5804.746} C_VEL
LIN {X 0,Y 199.92,Z 1174.569,A -85,B 0,C 180,E1 5799.628,E2 5799.628} C_VEL
LIN {X 0,Y 213.289,Z 1163.039,A -85,B 0,C 180,E1 5795.346,E2 5795.346} C_VEL
LIN {X 0,Y 226.962,Z 1150.356,A -85,B 0,C 180,E1 5791.762,E2 5791.762} C_VEL
LIN {X 0,Y 240.645,Z 1136.208,A -85,B 0,C 180,E1 5788.755,E2 5788.755} C_VEL
LIN {X 0,Y 254.934,Z 1119.935,A -85,B 0,C 180,E1 5786.085,E2 5786.085} C_VEL
LIN {X 0,Y 267.59,Z 1103.78,A -85,B 0,C 180,E1 5784.035,E2 5784.035} C_VEL
LIN {X 0,Y 280.707,Z 1084.874,A -85,B 0,C 180,E1 5782.166,E2 5782.166} C_VEL
LIN {X 0,Y 292.32,Z 1065.916,A -85,B 0,C 180,E1 5780.694,E2 5780.694} C_VEL
LIN {X 0,Y 302.915,Z 1045.675,A -85,B 0,C 180,E1 5779.475,E2 5779.475} C_VEL
LIN {X 0,Y 312.578,Z 1024.194,A -85,B 0,C 180,E1 5778.463,E2 5778.463} C_VEL
LIN {X 0,Y 320.162,Z 1003.997,A -85,B 0,C 180,E1 5777.73,E2 5777.73} C_VEL
LIN {X 0,Y 327.316,Z 980.477,A -85,B 0,C 180,E1 5777.091,E2 5777.091} C_VEL
LIN {X 0,Y 332.664,Z 957.62,A -85,B 0,C 180,E1 5776.62,E2 5776.62} C_VEL
LIN {X 0,Y 336.269,Z 934.283,A -85,B 0,C 180,E1 5776.229,E2 5776.229} C_VEL
LIN {X 0,Y 352.104,Z 784.623,A -85,B 0,C 180,E1 5774.094,E2 5774.094} C_VEL
LIN {X 0,Y 350.194,Z 777.929,A -85,B 0,C 180,E1 5771.446,E2 5771.446} C_VEL
LIN {X 0,Y 348.927,Z 773.211,A -85,B 0,C 180,E1 5768.985,E2 5768.985} C_VEL
LIN {X 0,Y 348.107,Z 769.926,A -85,B 0,C 180,E1 5766.432,E2 5766.432} C_VEL
LIN {X 0,Y 347.853,Z 768.018,A -85,B 0,C 180,E1 5764.451,E2 5764.451} C_VEL
LIN {X 0,Y 348.252,Z 767.129,A -85,B 0,C 180,E1 5760.494,E2 5760.494} C_VEL
LIN {X 0,Y 349.239,Z 768.246,A -85,B 0,C 180,E1 5757.867,E2 5757.867} C_VEL
LIN {X 0,Y 350.308,Z 769.783,A -85,B 0,C 180,E1 5755.99,E2 5755.99} C_VEL
LIN {X 0,Y 352.223,Z 773.384,A -85,B 0,C 180,E1 5753.398,E2 5753.398} C_VEL
LIN {X 0,Y 353.438,Z 775.989,A -85,B 0,C 180,E1 5752.034,E2 5752.034} C_VEL
LIN {X 0,Y 338.901,Z 909.337,A -85,B 0,C 180,E1 5750.073,E2 5750.073} C_VEL
LIN {X 0,Y 337.857,Z 917.028,A -85,B 0,C 180,E1 5750.12,E2 5750.12} C_VEL
LIN {X 0,Y 333.952,Z 937.47,A -85,B 0,C 180,E1 5750.858,E2 5750.858} C_VEL
LIN {X 0,Y 332.67,Z 944.013,A -85,B 0,C 180,E1 5750.862,E2 5750.862} C_VEL
LIN {X 0,Y 327.933,Z 967.302,A -85,B 0,C 180,E1 5750.387,E2 5750.387} C_VEL
LIN {X 0,Y 321.577,Z 990.078,A -85,B 0,C 180,E1 5749.759,E2 5749.759} C_VEL
LIN {X 0,Y 314.05,Z 1012.002,A -85,B 0,C 180,E1 5748.987,E2 5748.987} C_VEL
LIN {X 0,Y 305.543,Z 1032.32,A -85,B 0,C 180,E1 5748.082,E2 5748.082} C_VEL
LIN {X 0,Y 294.968,Z 1053.958,A -85,B 0,C 180,E1 5746.872,E2 5746.872} C_VEL
LIN {X 0,Y 284.38,Z 1072.582,A -85,B 0,C 180,E1 5745.571,E2 5745.571} C_VEL
LIN {X 0,Y 271.248,Z 1092.845,A -85,B 0,C 180,E1 5743.789,E2 5743.789} C_VEL
LIN {X 0,Y 258.772,Z 1109.884,A -85,B 0,C 180,E1 5741.898,E2 5741.898} C_VEL
LIN {X 0,Y 244.526,Z 1127.202,A -85,B 0,C 180,E1 5739.451,E2 5739.451} C_VEL
LIN {X 0,Y 230.769,Z 1142.375,A -85,B 0,C 180,E1 5736.713,E2 5736.713} C_VEL
LIN {X 0,Y 216.063,Z 1156.967,A -85,B 0,C 180,E1 5733.269,E2 5733.269} C_VEL
LIN {X 0,Y 201.523,Z 1170.327,A -85,B 0,C 180,E1 5729.131,E2 5729.131} C_VEL
LIN {X 0,Y 188.127,Z 1181.622,A -85,B 0,C 180,E1 5724.406,E2 5724.406} C_VEL
LIN {X 0,Y 174.991,Z 1192.197,A -85,B 0,C 180,E1 5718.461,E2 5718.461} C_VEL
LIN {X 0,Y 164.322,Z 1200.478,A -85,B 0,C 180,E1 5712.014,E2 5712.014} C_VEL
LIN {X 0,Y 154.72,Z 1208.049,A -85,B 0,C 180,E1 5703.763,E2 5703.763} C_VEL
LIN {X 0,Y 148.761,Z 1213.166,A -85,B 0,C 180,E1 5695.753,E2 5695.753} C_VEL
LIN {X 0,Y 145.062,Z 1217.099,A -85,B 0,C 180,E1 5686.415,E2 5686.415} C_VEL
LIN {X 0,Y 144.039,Z 1218.98,A -85,B 0,C 180,E1 5678.784,E2 5678.784} C_VEL
LIN {X 0,Y 143.998,Z 1219.67,A -85,B 0,C 180,E1 5672.786,E2 5672.786} C_VEL
LIN {X 0,Y 144.002,Z 1219.688,A -85,B 0,C 180,E1 5667.612,E2 5667.612} C_VEL
LIN {X 0,Y 144.019,Z 1219.033,A -85,B 0,C 180,E1 5661.617,E2 5661.617} C_VEL
LIN {X 0,Y 144.878,Z 1217.307,A -85,B 0,C 180,E1 5654.386,E2 5654.386} C_VEL
LIN {X 0,Y 147.995,Z 1213.896,A -85,B 0,C 180,E1 5645.662,E2 5645.662} C_VEL
LIN {X 0,Y 153.723,Z 1208.774,A -85,B 0,C 180,E1 5637.326,E2 5637.326} C_VEL
LIN {X 0,Y 162.514,Z 1201.837,A -85,B 0,C 180,E1 5629.296,E2 5629.296} C_VEL
LIN {X 0,Y 173.181,Z 1193.452,A -85,B 0,C 180,E1 5622.495,E2 5622.495} C_VEL
LIN {X 0,Y 186.218,Z 1183.06,A -85,B 0,C 180,E1 5616.352,E2 5616.352} C_VEL
LIN {X 0,Y 199.425,Z 1171.925,A -85,B 0,C 180,E1 5611.534,E2 5611.534} C_VEL
LIN {X 0,Y 214.549,Z 1158.19,A -85,B 0,C 180,E1 5607.113,E2 5607.113} C_VEL
LIN {X 0,Y 228.743,Z 1144.217,A -85,B 0,C 180,E1 5603.713,E2 5603.713} C_VEL
LIN {X 0,Y 242.864,Z 1128.799,A -85,B 0,C 180,E1 5600.845,E2 5600.845} C_VEL
LIN {X 0,Y 257.059,Z 1111.795,A -85,B 0,C 180,E1 5598.366,E2 5598.366} C_VEL
LIN {X 0,Y 270.352,Z 1093.705,A -85,B 0,C 180,E1 5596.325,E2 5596.325} C_VEL
LIN {X 0,Y 283.08,Z 1074.268,A -85,B 0,C 180,E1 5594.583,E2 5594.583} C_VEL
LIN {X 0,Y 293.782,Z 1055.575,A -85,B 0,C 180,E1 5593.252,E2 5593.252} C_VEL
LIN {X 0,Y 304.62,Z 1033.712,A -85,B 0,C 180,E1 5592.006,E2 5592.006} C_VEL
LIN {X 0,Y 312.832,Z 1014.271,A -85,B 0,C 180,E1 5591.123,E2 5591.123} C_VEL
LIN {X 0,Y 320.869,Z 991.362,A -85,B 0,C 180,E1 5590.294,E2 5590.294} C_VEL
LIN {X 0,Y 327.202,Z 968.921,A -85,B 0,C 180,E1 5589.665,E2 5589.665} C_VEL
LIN {X 0,Y 332.116,Z 945.379,A -85,B 0,C 180,E1 5589.174,E2 5589.174} C_VEL
LIN {X 0,Y 335.664,Z 920.589,A -85,B 0,C 180,E1 5588.777,E2 5588.777} C_VEL
LIN {X 0,Y 351.03,Z 781.521,A -85,B 0,C 180,E1 5586.752,E2 5586.752} C_VEL
LIN {X 0,Y 349.364,Z 778.313,A -85,B 0,C 180,E1 5584.596,E2 5584.596} C_VEL
LIN {X 0,Y 348.363,Z 776.493,A -85,B 0,C 180,E1 5582.961,E2 5582.961} C_VEL
LIN {X 0,Y 347.039,Z 774.716,A -85,B 0,C 180,E1 5579.835,E2 5579.835} C_VEL
LIN {X 0,Y 346.502,Z 775.175,A -85,B 0,C 180,E1 5576.691,E2 5576.691} C_VEL
LIN {X 0,Y 346.579,Z 776.141,A -85,B 0,C 180,E1 5574.869,E2 5574.869} C_VEL
LIN {X 0,Y 347.171,Z 779.586,A -85,B 0,C 180,E1 5571.97,E2 5571.97} C_VEL
LIN {X 0,Y 347.985,Z 782.812,A -85,B 0,C 180,E1 5569.989,E2 5569.989} C_VEL
LIN {X 0,Y 349.643,Z 789.14,A -85,B 0,C 180,E1 5567.223,E2 5567.223} C_VEL
LIN {X 0,Y 349.77,Z 789.976,A -85,B 0,C 180,E1 5567.004,E2 5567.004} C_VEL
LIN {X 0,Y 333.413,Z 940.319,A -85,B 0,C 180,E1 5564.914,E2 5564.914} C_VEL
LIN {X 0,Y 329.133,Z 963.885,A -85,B 0,C 180,E1 5564.507,E2 5564.507} C_VEL
LIN {X 0,Y 323.435,Z 986.573,A -85,B 0,C 180,E1 5564.031,E2 5564.031} C_VEL
LIN {X 0,Y 316.575,Z 1007.498,A -85,B 0,C 180,E1 5563.448,E2 5563.448} C_VEL
LIN {X 0,Y 307.972,Z 1029.291,A -85,B 0,C 180,E1 5562.648,E2 5562.648} C_VEL
LIN {X 0,Y 298.563,Z 1049.195,A -85,B 0,C 180,E1 5561.698,E2 5561.698} C_VEL
LIN {X 0,Y 287.058,Z 1070.04,A -85,B 0,C 180,E1 5560.421,E2 5560.421} C_VEL
LIN {X 0,Y 275.306,Z 1088.612,A -85,B 0,C 180,E1 5558.967,E2 5558.967} C_VEL
LIN {X 0,Y 262.483,Z 1106.252,A -85,B 0,C 180,E1 5557.195,E2 5557.195} C_VEL
LIN {X 0,Y 248.931,Z 1122.971,A -85,B 0,C 180,E1 5555.054,E2 5555.054} C_VEL
LIN {X 0,Y 235.397,Z 1137.746,A -85,B 0,C 180,E1 5552.59,E2 5552.59} C_VEL
LIN {X 0,Y 220.649,Z 1152.355,A -85,B 0,C 180,E1 5549.426,E2 5549.426} C_VEL
LIN {X 0,Y 206.676,Z 1164.85,A -85,B 0,C 180,E1 5545.819,E2 5545.819} C_VEL
LIN {X 0,Y 192.324,Z 1176.57,A -85,B 0,C 180,E1 5541.244,E2 5541.244} C_VEL
LIN {X 0,Y 179.373,Z 1186.449,A -85,B 0,C 180,E1 5535.978,E2 5535.978} C_VEL
LIN {X 0,Y 167.593,Z 1194.773,A -85,B 0,C 180,E1 5529.67,E2 5529.67} C_VEL
LIN {X 0,Y 157.624,Z 1201.714,A -85,B 0,C 180,E1 5522.197,E2 5522.197} C_VEL
LIN {X 0,Y 150.622,Z 1206.639,A -85,B 0,C 180,E1 5514.303,E2 5514.303} C_VEL
LIN {X 0,Y 145.989,Z 1210.253,A -85,B 0,C 180,E1 5505.044,E2 5505.044} C_VEL
LIN {X 0,Y 144.352,Z 1211.926,A -85,B 0,C 180,E1 5497.162,E2 5497.162} C_VEL
LIN {X 0,Y 144.062,Z 1212.455,A -85,B 0,C 180,E1 5489.602,E2 5489.602} C_VEL
LIN {X 0,Y 144.457,Z 1211.794,A -85,B 0,C 180,E1 5481.814,E2 5481.814} C_VEL
LIN {X 0,Y 146.378,Z 1209.975,A -85,B 0,C 180,E1 5473.736,E2 5473.736} C_VEL
LIN {X 0,Y 151.096,Z 1206.344,A -85,B 0,C 180,E1 5464.944,E2 5464.944} C_VEL
LIN {X 0,Y 158.704,Z 1201.098,A -85,B 0,C 180,E1 5456.762,E2 5456.762} C_VEL
LIN {X 0,Y 168.488,Z 1194.26,A -85,B 0,C 180,E1 5449.696,E2 5449.696} C_VEL
LIN {X 0,Y 180.758,Z 1185.524,A -85,B 0,C 180,E1 5443.309,E2 5443.309} C_VEL
LIN {X 0,Y 193.523,Z 1175.801,A -85,B 0,C 180,E1 5438.249,E2 5438.249} C_VEL
LIN {X 0,Y 207.991,Z 1163.901,A -85,B 0,C 180,E1 5433.732,E2 5433.732} C_VEL
LIN {X 0,Y 222.05,Z 1151.307,A -85,B 0,C 180,E1 5430.169,E2 5430.169} C_VEL
LIN {X 0,Y 236.073,Z 1137.315,A -85,B 0,C 180,E1 5427.199,E2 5427.199} C_VEL
LIN {X 0,Y 250.23,Z 1121.786,A -85,B 0,C 180,E1 5424.65,E2 5424.65} C_VEL
LIN {X 0,Y 263.636,Z 1105.127,A -85,B 0,C 180,E1 5422.558,E2 5422.558} C_VEL
LIN {X 0,Y 277.352,Z 1085.929,A -85,B 0,C 180,E1 5420.69,E2 5420.69} C_VEL
LIN {X 0,Y 288.706,Z 1067.814,A -85,B 0,C 180,E1 5419.313,E2 5419.313} C_VEL
LIN {X 0,Y 299.788,Z 1047.346,A -85,B 0,C 180,E1 5418.097,E2 5418.097} C_VEL
LIN {X 0,Y 309.216,Z 1027.211,A -85,B 0,C 180,E1 5417.156,E2 5417.156} C_VEL
LIN {X 0,Y 317.374,Z 1006.125,A -85,B 0,C 180,E1 5416.403,E2 5416.403} C_VEL
LIN {X 0,Y 324.555,Z 983.653,A -85,B 0,C 180,E1 5415.796,E2 5415.796} C_VEL
LIN {X 0,Y 329.941,Z 961.646,A -85,B 0,C 180,E1 5415.349,E2 5415.349} C_VEL
LIN {X 0,Y 334.162,Z 936.976,A -85,B 0,C 180,E1 5414.934,E2 5414.934} C_VEL
LIN {X 0,Y 350.103,Z 789.891,A -85,B 0,C 180,E1 5412.872,E2 5412.872} C_VEL
LIN {X 0,Y 348.671,Z 784.488,A -85,B 0,C 180,E1 5410.576,E2 5410.576} C_VEL
LIN {X 0,Y 347.713,Z 780.575,A -85,B 0,C 180,E1 5408.433,E2 5408.433} C_VEL
LIN {X 0,Y 347.063,Z 777.651,A -85,B 0,C 180,E1 5406.119,E2 5406.119} C_VEL
LIN {X 0,Y 346.864,Z 775.915,A -85,B 0,C 180,E1 5404.298,E2 5404.298} C_VEL
LIN {X 0,Y 347.261,Z 775.068,A -85,B 0,C 180,E1 5400.495,E2 5400.495} C_VEL
LIN {X 0,Y 348.244,Z 776.225,A -85,B 0,C 180,E1 5397.861,E2 5397.861} C_VEL
LIN {X 0,Y 349.249,Z 777.788,A -85,B 0,C 180,E1 5396.06,E2 5396.06} C_VEL
LIN {X 0,Y 351.006,Z 781.194,A -85,B 0,C 180,E1 5393.621,E2 5393.621} C_VEL
LIN {X 0,Y 351.306,Z 782.052,A -85,B 0,C 180,E1 5393.229,E2 5393.229} C_VEL
LIN {X 0,Y 334.16,Z 934.81,A -85,B 0,C 180,E1 5391.016,E2 5391.016} C_VEL
LIN {X 0,Y 332.67,Z 944.013,A -85,B 0,C 180,E1 5390.862,E2 5390.862} C_VEL
LIN {X 0,Y 331.112,Z 951.61,A -85,B 0,C 180,E1 5390.918,E2 5390.918} C_VEL
LIN {X 0,Y 325.62,Z 970.646,A -85,B 0,C 180,E1 5391.545,E2 5391.545} C_VEL
LIN {X 0,Y 323.458,Z 978.1,A -85,B 0,C 180,E1 5391.501,E2 5391.501} C_VEL
LIN {X 0,Y 316.021,Z 1001.74,A -85,B 0,C 180,E1 5390.798,E2 5390.798} C_VEL
LIN {X 0,Y 308.126,Z 1022.266,A -85,B 0,C 180,E1 5390.012,E2 5390.012} C_VEL
LIN {X 0,Y 298.306,Z 1043.559,A -85,B 0,C 180,E1 5388.985,E2 5388.985} C_VEL
LIN {X 0,Y 287.482,Z 1063.821,A -85,B 0,C 180,E1 5387.771,E2 5387.771} C_VEL
LIN {X 0,Y 275.754,Z 1082.649,A -85,B 0,C 180,E1 5386.346,E2 5386.346} C_VEL
LIN {X 0,Y 262.894,Z 1101.083,A -85,B 0,C 180,E1 5384.607,E2 5384.607} C_VEL
LIN {X 0,Y 249.419,Z 1118,A -85,B 0,C 180,E1 5382.569,E2 5382.569} C_VEL
LIN {X 0,Y 235.046,Z 1134.344,A -85,B 0,C 180,E1 5380.069,E2 5380.069} C_VEL
LIN {X 0,Y 220.353,Z 1149.263,A -85,B 0,C 180,E1 5377.09,E2 5377.09} C_VEL
LIN {X 0,Y 204.052,Z 1164.289,A -85,B 0,C 180,E1 5373.1,E2 5373.1} C_VEL
LIN {X 0,Y 190.253,Z 1175.961,A -85,B 0,C 180,E1 5368.94,E2 5368.94} C_VEL
LIN {X 0,Y 175.653,Z 1187.384,A -85,B 0,C 180,E1 5363.38,E2 5363.38} C_VEL
LIN {X 0,Y 162.876,Z 1196.97,A -85,B 0,C 180,E1 5356.929,E2 5356.929} C_VEL
LIN {X 0,Y 152.284,Z 1204.601,A -85,B 0,C 180,E1 5349.559,E2 5349.559} C_VEL
LIN {X 0,Y 143.932,Z 1210.931,A -85,B 0,C 180,E1 5340.934,E2 5340.934} C_VEL
LIN {X 0,Y 138.963,Z 1215.097,A -85,B 0,C 180,E1 5332.417,E2 5332.417} C_VEL
LIN {X 0,Y 136.419,Z 1218.093,A -85,B 0,C 180,E1 5323.133,E2 5323.133} C_VEL
LIN {X 0,Y 135.978,Z 1219.34,A -85,B 0,C 180,E1 5315.062,E2 5315.062} C_VEL
LIN {X 0,Y 136.023,Z 1219.552,A -85,B 0,C 180,E1 5308.666,E2 5308.666} C_VEL
LIN {X 0,Y 136.006,Z 1218.972,A -85,B 0,C 180,E1 5301.971,E2 5301.971} C_VEL
LIN {X 0,Y 136.954,Z 1217.219,A -85,B 0,C 180,E1 5293.893,E2 5293.893} C_VEL
LIN {X 0,Y 140.332,Z 1213.875,A -85,B 0,C 180,E1 5284.691,E2 5284.691} C_VEL
LIN {X 0,Y 146.492,Z 1208.823,A -85,B 0,C 180,E1 5275.966,E2 5275.966} C_VEL
LIN {X 0,Y 155.854,Z 1201.979,A -85,B 0,C 180,E1 5267.654,E2 5267.654} C_VEL
LIN {X 0,Y 167.276,Z 1193.526,A -85,B 0,C 180,E1 5260.614,E2 5260.614} C_VEL
LIN {X 0,Y 180.764,Z 1183.352,A -85,B 0,C 180,E1 5254.496,E2 5254.496} C_VEL
LIN {X 0,Y 193.776,Z 1172.858,A -85,B 0,C 180,E1 5249.905,E2 5249.905} C_VEL
LIN {X 0,Y 209.359,Z 1159.359,A -85,B 0,C 180,E1 5245.494,E2 5245.494} C_VEL
LIN {X 0,Y 223.549,Z 1145.877,A -85,B 0,C 180,E1 5242.205,E2 5242.205} C_VEL
LIN {X 0,Y 239.209,Z 1129.435,A -85,B 0,C 180,E1 5239.153,E2 5239.153} C_VEL
LIN {X 0,Y 253.283,Z 1113.042,A -85,B 0,C 180,E1 5236.806,E2 5236.806} C_VEL
LIN {X 0,Y 266.839,Z 1095.163,A -85,B 0,C 180,E1 5234.82,E2 5234.82} C_VEL
LIN {X 0,Y 279.778,Z 1076.042,A -85,B 0,C 180,E1 5233.133,E2 5233.133} C_VEL
LIN {X 0,Y 291.102,Z 1056.706,A -85,B 0,C 180,E1 5231.792,E2 5231.792} C_VEL
LIN {X 0,Y 302.105,Z 1035.091,A -85,B 0,C 180,E1 5230.593,E2 5230.593} C_VEL
LIN {X 0,Y 310.432,Z 1015.804,A -85,B 0,C 180,E1 5229.741,E2 5229.741} C_VEL
LIN {X 0,Y 318.813,Z 992.561,A -85,B 0,C 180,E1 5228.923,E2 5228.923} C_VEL
LIN {X 0,Y 325.071,Z 970.865,A -85,B 0,C 180,E1 5228.331,E2 5228.331} C_VEL
LIN {X 0,Y 330.295,Z 946.793,A -85,B 0,C 180,E1 5227.839,E2 5227.839} C_VEL
LIN {X 0,Y 333.86,Z 922.961,A -85,B 0,C 180,E1 5227.466,E2 5227.466} C_VEL
LIN {X 0,Y 349.038,Z 787.652,A -85,B 0,C 180,E1 5225.548,E2 5225.548} C_VEL
LIN {X 0,Y 347.369,Z 784.474,A -85,B 0,C 180,E1 5222.97,E2 5222.97} C_VEL
LIN {X 0,Y 346.058,Z 782.659,A -85,B 0,C 180,E1 5219.834,E2 5219.834} C_VEL
LIN {X 0,Y 345.526,Z 783.136,A -85,B 0,C 180,E1 5216.682,E2 5216.682} C_VEL
LIN {X 0,Y 345.581,Z 784.045,A -85,B 0,C 180,E1 5215.02,E2 5215.02} C_VEL
LIN {X 0,Y 346.098,Z 787.408,A -85,B 0,C 180,E1 5212.196,E2 5212.196} C_VEL
LIN {X 0,Y 346.828,Z 790.553,A -85,B 0,C 180,E1 5210.29,E2 5210.29} C_VEL
LIN {X 0,Y 347.93,Z 795.077,A -85,B 0,C 180,E1 5208.237,E2 5208.237} C_VEL
LIN {X 0,Y 331.856,Z 939.982,A -85,B 0,C 180,E1 5206.271,E2 5206.271} C_VEL
LIN {X 0,Y 327.536,Z 963.488,A -85,B 0,C 180,E1 5205.881,E2 5205.881} C_VEL
LIN {X 0,Y 321.802,Z 986.13,A -85,B 0,C 180,E1 5205.431,E2 5205.431} C_VEL
LIN {X 0,Y 314.86,Z 1007.083,A -85,B 0,C 180,E1 5204.877,E2 5204.877} C_VEL
LIN {X 0,Y 306.146,Z 1028.933,A -85,B 0,C 180,E1 5204.116,E2 5204.116} C_VEL
LIN {X 0,Y 296.604,Z 1048.865,A -85,B 0,C 180,E1 5203.209,E2 5203.209} C_VEL
LIN {X 0,Y 284.923,Z 1069.76,A -85,B 0,C 180,E1 5201.989,E2 5201.989} C_VEL
LIN {X 0,Y 272.97,Z 1088.357,A -85,B 0,C 180,E1 5200.595,E2 5200.595} C_VEL
LIN {X 0,Y 259.906,Z 1106.044,A -85,B 0,C 180,E1 5198.891,E2 5198.891} C_VEL
LIN {X 0,Y 246.704,Z 1122.09,A -85,B 0,C 180,E1 5196.926,E2 5196.926} C_VEL
LIN {X 0,Y 232.607,Z 1137.19,A -85,B 0,C 180,E1 5194.513,E2 5194.513} C_VEL
LIN {X 0,Y 218.214,Z 1151.224,A -85,B 0,C 180,E1 5191.612,E2 5191.612} C_VEL
LIN {X 0,Y 203.717,Z 1163.84,A -85,B 0,C 180,E1 5188.113,E2 5188.113} C_VEL
LIN {X 0,Y 188.356,Z 1176.053,A -85,B 0,C 180,E1 5183.519,E2 5183.519} C_VEL
LIN {X 0,Y 175.052,Z 1185.774,A -85,B 0,C 180,E1 5178.438,E2 5178.438} C_VEL
LIN {X 0,Y 162.468,Z 1194.3,A -85,B 0,C 180,E1 5172.129,E2 5172.129} C_VEL
LIN {X 0,Y 152.053,Z 1201.177,A -85,B 0,C 180,E1 5164.896,E2 5164.896} C_VEL
LIN {X 0,Y 143.851,Z 1206.449,A -85,B 0,C 180,E1 5156.413,E2 5156.413} C_VEL
LIN {X 0,Y 138.521,Z 1210.231,A -85,B 0,C 180,E1 5146.781,E2 5146.781} C_VEL
LIN {X 0,Y 136.488,Z 1212.002,A -85,B 0,C 180,E1 5138.425,E2 5138.425} C_VEL
LIN {X 0,Y 136.066,Z 1212.648,A -85,B 0,C 180,E1 5130.421,E2 5130.421} C_VEL
LIN {X 0,Y 136.384,Z 1212.166,A -85,B 0,C 180,E1 5122.417,E2 5122.417} C_VEL
LIN {X 0,Y 138.199,Z 1210.506,A -85,B 0,C 180,E1 5114.042,E2 5114.042} C_VEL
LIN {X 0,Y 142.95,Z 1207.15,A -85,B 0,C 180,E1 5104.744,E2 5104.744} C_VEL
LIN {X 0,Y 150.345,Z 1202.294,A -85,B 0,C 180,E1 5096.497,E2 5096.497} C_VEL
LIN {X 0,Y 161.338,Z 1195.161,A -85,B 0,C 180,E1 5088.463,E2 5088.463} C_VEL
LIN {X 0,Y 173.73,Z 1186.876,A -85,B 0,C 180,E1 5082.062,E2 5082.062} C_VEL
LIN {X 0,Y 187.636,Z 1176.747,A -85,B 0,C 180,E1 5076.644,E2 5076.644} C_VEL
LIN {X 0,Y 202.867,Z 1164.765,A -85,B 0,C 180,E1 5072.035,E2 5072.035} C_VEL
LIN {X 0,Y 216.535,Z 1152.934,A -85,B 0,C 180,E1 5068.678,E2 5068.678} C_VEL
LIN {X 0,Y 231.888,Z 1138.212,A -85,B 0,C 180,E1 5065.544,E2 5065.544} C_VEL
LIN {X 0,Y 246.593,Z 1122.536,A -85,B 0,C 180,E1 5063.014,E2 5063.014} C_VEL
LIN {X 0,Y 260.227,Z 1106.008,A -85,B 0,C 180,E1 5060.987,E2 5060.987} C_VEL
LIN {X 0,Y 273.302,Z 1088.313,A -85,B 0,C 180,E1 5059.287,E2 5059.287} C_VEL
LIN {X 0,Y 284.818,Z 1070.438,A -85,B 0,C 180,E1 5057.946,E2 5057.946} C_VEL
LIN {X 0,Y 296.501,Z 1049.684,A -85,B 0,C 180,E1 5056.724,E2 5056.724} C_VEL
LIN {X 0,Y 306.121,Z 1029.672,A -85,B 0,C 180,E1 5055.809,E2 5055.809} C_VEL
LIN {X 0,Y 314.758,Z 1008.251,A -85,B 0,C 180,E1 5055.054,E2 5055.054} C_VEL
LIN {X 0,Y 321.933,Z 986.733,A -85,B 0,C 180,E1 5054.481,E2 5054.481} C_VEL
LIN {X 0,Y 327.786,Z 963.83,A -85,B 0,C 180,E1 5054.024,E2 5054.024} C_VEL
LIN {X 0,Y 332.153,Z 940.233,A -85,B 0,C 180,E1 5053.632,E2 5053.632} C_VEL
LIN {X 0,Y 348.253,Z 795.281,A -85,B 0,C 180,E1 5051.641,E2 5051.641} C_VEL
LIN {X 0,Y 346.804,Z 788.957,A -85,B 0,C 180,E1 5048.623,E2 5048.623} C_VEL
LIN {X 0,Y 346.047,Z 785.546,A -85,B 0,C 180,E1 5045.971,E2 5045.971} C_VEL
LIN {X 0,Y 345.876,Z 783.812,A -85,B 0,C 180,E1 5044.145,E2 5044.145} C_VEL
LIN {X 0,Y 346.317,Z 783.031,A -85,B 0,C 180,E1 5040.331,E2 5040.331} C_VEL
LIN {X 0,Y 347.502,Z 784.532,A -85,B 0,C 180,E1 5037.361,E2 5037.361} C_VEL
LIN {X 0,Y 349.192,Z 787.602,A -85,B 0,C 180,E1 5034.66,E2 5034.66} C_VEL
LIN {X 0,Y 349.324,Z 788.181,A -85,B 0,C 180,E1 5034.439,E2 5034.439} C_VEL
LIN {X 0,Y 332.559,Z 935.191,A -85,B 0,C 180,E1 5032.362,E2 5032.362} C_VEL
LIN {X 0,Y 328.14,Z 959.181,A -85,B 0,C 180,E1 5031.93,E2 5031.93} C_VEL
LIN {X 0,Y 323.458,Z 978.1,A -85,B 0,C 180,E1 5031.501,E2 5031.501} C_VEL
LIN {X 0,Y 321.21,Z 985.551,A -85,B 0,C 180,E1 5031.472,E2 5031.472} C_VEL
LIN {X 0,Y 314.011,Z 1004.121,A -85,B 0,C 180,E1 5031.979,E2 5031.979} C_VEL
LIN {X 0,Y 311.038,Z 1011.266,A -85,B 0,C 180,E1 5031.906,E2 5031.906} C_VEL
LIN {X 0,Y 301.945,Z 1032.439,A -85,B 0,C 180,E1 5031.046,E2 5031.046} C_VEL
LIN {X 0,Y 291.409,Z 1053.451,A -85,B 0,C 180,E1 5029.973,E2 5029.973} C_VEL
LIN {X 0,Y 280.334,Z 1072.352,A -85,B 0,C 180,E1 5028.764,E2 5028.764} C_VEL
LIN {X 0,Y 266.677,Z 1092.717,A -85,B 0,C 180,E1 5027.115,E2 5027.115} C_VEL
LIN {X 0,Y 254.003,Z 1109.369,A -85,B 0,C 180,E1 5025.408,E2 5025.408} C_VEL
LIN {X 0,Y 239.235,Z 1126.603,A -85,B 0,C 180,E1 5023.152,E2 5023.152} C_VEL
LIN {X 0,Y 224.745,Z 1141.807,A -85,B 0,C 180,E1 5020.588,E2 5020.588} C_VEL
LIN {X 0,Y 209.136,Z 1156.459,A -85,B 0,C 180,E1 5017.325,E2 5017.325} C_VEL
LIN {X 0,Y 193.53,Z 1169.855,A -85,B 0,C 180,E1 5013.353,E2 5013.353} C_VEL
LIN {X 0,Y 178.268,Z 1181.685,A -85,B 0,C 180,E1 5008.487,E2 5008.487} C_VEL
LIN {X 0,Y 163.217,Z 1192.589,A -85,B 0,C 180,E1 5002.208,E2 5002.208} C_VEL
LIN {X 0,Y 151.36,Z 1200.769,A -85,B 0,C 180,E1 4995.514,E2 4995.514} C_VEL
LIN {X 0,Y 140.882,Z 1207.89,A -85,B 0,C 180,E1 4987.103,E2 4987.103} C_VEL
LIN {X 0,Y 133.641,Z 1213.147,A -85,B 0,C 180,E1 4978.01,E2 4978.01} C_VEL
LIN {X 0,Y 129.375,Z 1216.803,A -85,B 0,C 180,E1 4968.007,E2 4968.007} C_VEL
LIN {X 0,Y 128.076,Z 1218.64,A -85,B 0,C 180,E1 4959.436,E2 4959.436} C_VEL
LIN {X 0,Y 128.002,Z 1219.286,A -85,B 0,C 180,E1 4952.686,E2 4952.686} C_VEL
LIN {X 0,Y 128.002,Z 1219.279,A -85,B 0,C 180,E1 4947.314,E2 4947.314} C_VEL
LIN {X 0,Y 128.076,Z 1218.62,A -85,B 0,C 180,E1 4940.564,E2 4940.564} C_VEL
LIN {X 0,Y 129.375,Z 1216.769,A -85,B 0,C 180,E1 4931.993,E2 4931.993} C_VEL
LIN {X 0,Y 133.959,Z 1212.821,A -85,B 0,C 180,E1 4921.465,E2 4921.465} C_VEL
LIN {X 0,Y 140.878,Z 1207.813,A -85,B 0,C 180,E1 4912.895,E2 4912.895} C_VEL
LIN {X 0,Y 151.868,Z 1200.296,A -85,B 0,C 180,E1 4904.141,E2 4904.141} C_VEL
LIN {X 0,Y 163.822,Z 1192.052,A -85,B 0,C 180,E1 4897.493,E2 4897.493} C_VEL
LIN {X 0,Y 178.259,Z 1181.532,A -85,B 0,C 180,E1 4891.508,E2 4891.508} C_VEL
LIN {X 0,Y 192.976,Z 1170.105,A -85,B 0,C 180,E1 4886.794,E2 4886.794} C_VEL
LIN {X 0,Y 208.321,Z 1156.95,A -85,B 0,C 180,E1 4882.85,E2 4882.85} C_VEL
LIN {X 0,Y 223.894,Z 1142.399,A -85,B 0,C 180,E1 4879.563,E2 4879.563} C_VEL
LIN {X 0,Y 238.356,Z 1127.248,A -85,B 0,C 180,E1 4876.978,E2 4876.978} C_VEL
LIN {X 0,Y 253.24,Z 1109.961,A -85,B 0,C 180,E1 4874.688,E2 4874.688} C_VEL
LIN {X 0,Y 266.212,Z 1092.929,A -85,B 0,C 180,E1 4872.929,E2 4872.929} C_VEL
LIN {X 0,Y 279.862,Z 1072.6,A -85,B 0,C 180,E1 4871.275,E2 4871.275} C_VEL
LIN {X 0,Y 290.933,Z 1053.728,A -85,B 0,C 180,E1 4870.061,E2 4870.061} C_VEL
LIN {X 0,Y 301.644,Z 1032.398,A -85,B 0,C 180,E1 4868.968,E2 4868.968} C_VEL
LIN {X 0,Y 310.782,Z 1011.093,A -85,B 0,C 180,E1 4868.102,E2 4868.102} C_VEL
LIN {X 0,Y 318.126,Z 990.017,A -85,B 0,C 180,E1 4867.43,E2 4867.43} C_VEL
LIN {X 0,Y 324.578,Z 967.324,A -85,B 0,C 180,E1 4866.859,E2 4866.859} C_VEL
LIN {X 0,Y 329.37,Z 944.26,A -85,B 0,C 180,E1 4866.425,E2 4866.425} C_VEL
LIN {X 0,Y 333.372,Z 915.256,A -85,B 0,C 180,E1 4865.999,E2 4865.999} C_VEL
LIN {X 0,Y 347.156,Z 794.143,A -85,B 0,C 180,E1 4864.332,E2 4864.332} C_VEL
LIN {X 0,Y 346.192,Z 792.234,A -85,B 0,C 180,E1 4862.649,E2 4862.649} C_VEL
LIN {X 0,Y 345.036,Z 790.572,A -85,B 0,C 180,E1 4859.668,E2 4859.668} C_VEL
LIN {X 0,Y 344.546,Z 791.228,A -85,B 0,C 180,E1 4856.339,E2 4856.339} C_VEL
LIN {X 0,Y 344.591,Z 792.134,A -85,B 0,C 180,E1 4855.006,E2 4855.006} C_VEL
LIN {X 0,Y 345.054,Z 795.348,A -85,B 0,C 180,E1 4852.34,E2 4852.34} C_VEL
LIN {X 0,Y 345.717,Z 798.467,A -85,B 0,C 180,E1 4850.511,E2 4850.511} C_VEL
LIN {X 0,Y 346.195,Z 800.714,A -85,B 0,C 180,E1 4849.473,E2 4849.473} C_VEL
LIN {X 0,Y 330.473,Z 939.752,A -85,B 0,C 180,E1 4847.639,E2 4847.639} C_VEL
LIN {X 0,Y 326.1,Z 963.218,A -85,B 0,C 180,E1 4847.266,E2 4847.266} C_VEL
LIN {X 0,Y 320.363,Z 985.679,A -85,B 0,C 180,E1 4846.844,E2 4846.844} C_VEL
LIN {X 0,Y 313.343,Z 1006.667,A -85,B 0,C 180,E1 4846.321,E2 4846.321} C_VEL
LIN {X 0,Y 304.524,Z 1028.575,A -85,B 0,C 180,E1 4845.601,E2 4845.601} C_VEL
LIN {X 0,Y 294.855,Z 1048.534,A -85,B 0,C 180,E1 4844.74,E2 4844.74} C_VEL
LIN {X 0,Y 283.071,Z 1069.373,A -85,B 0,C 180,E1 4843.585,E2 4843.585} C_VEL
LIN {X 0,Y 271.306,Z 1087.44,A -85,B 0,C 180,E1 4842.3,E2 4842.3} C_VEL
LIN {X 0,Y 257.561,Z 1105.836,A -85,B 0,C 180,E1 4840.618,E2 4840.618} C_VEL
LIN {X 0,Y 243.662,Z 1122.397,A -85,B 0,C 180,E1 4838.667,E2 4838.667} C_VEL
LIN {X 0,Y 229.252,Z 1137.47,A -85,B 0,C 180,E1 4836.332,E2 4836.332} C_VEL
LIN {X 0,Y 213.684,Z 1152.163,A -85,B 0,C 180,E1 4833.344,E2 4833.344} C_VEL
LIN {X 0,Y 199.559,Z 1164.084,A -85,B 0,C 180,E1 4830.087,E2 4830.087} C_VEL
LIN {X 0,Y 183.274,Z 1176.547,A -85,B 0,C 180,E1 4825.431,E2 4825.431} C_VEL
LIN {X 0,Y 169.136,Z 1186.448,A -85,B 0,C 180,E1 4820.22,E2 4820.22} C_VEL
LIN {X 0,Y 155.988,Z 1194.859,A -85,B 0,C 180,E1 4813.809,E2 4813.809} C_VEL
LIN {X 0,Y 145.024,Z 1201.64,A -85,B 0,C 180,E1 4806.364,E2 4806.364} C_VEL
LIN {X 0,Y 136.643,Z 1206.659,A -85,B 0,C 180,E1 4797.924,E2 4797.924} C_VEL
LIN {X 0,Y 130.812,Z 1210.438,A -85,B 0,C 180,E1 4787.803,E2 4787.803} C_VEL
LIN {X 0,Y 128.546,Z 1212.21,A -85,B 0,C 180,E1 4778.932,E2 4778.932} C_VEL
LIN {X 0,Y 128.069,Z 1212.853,A -85,B 0,C 180,E1 4770.447,E2 4770.447} C_VEL
LIN {X 0,Y 128.431,Z 1212.371,A -85,B 0,C 180,E1 4761.944,E2 4761.944} C_VEL
LIN {X 0,Y 130.455,Z 1210.712,A -85,B 0,C 180,E1 4753.067,E2 4753.067} C_VEL
LIN {X 0,Y 135.667,Z 1207.359,A -85,B 0,C 180,E1 4743.284,E2 4743.284} C_VEL
LIN {X 0,Y 143.647,Z 1202.502,A -85,B 0,C 180,E1 4734.709,E2 4734.709} C_VEL
LIN {X 0,Y 155.352,Z 1195.374,A -85,B 0,C 180,E1 4726.476,E2 4726.476} C_VEL
LIN {X 0,Y 168.4,Z 1187.091,A -85,B 0,C 180,E1 4720.011,E2 4720.011} C_VEL
LIN {X 0,Y 182.528,Z 1177.246,A -85,B 0,C 180,E1 4714.73,E2 4714.73} C_VEL
LIN {X 0,Y 197.93,Z 1165.629,A -85,B 0,C 180,E1 4710.252,E2 4710.252} C_VEL
LIN {X 0,Y 212.774,Z 1153.179,A -85,B 0,C 180,E1 4706.768,E2 4706.768} C_VEL
LIN {X 0,Y 228.314,Z 1138.693,A -85,B 0,C 180,E1 4703.755,E2 4703.755} C_VEL
LIN {X 0,Y 242.698,Z 1123.74,A -85,B 0,C 180,E1 4701.399,E2 4701.399} C_VEL
LIN {X 0,Y 257.02,Z 1106.888,A -85,B 0,C 180,E1 4699.375,E2 4699.375} C_VEL
LIN {X 0,Y 270.177,Z 1089.561,A -85,B 0,C 180,E1 4697.754,E2 4697.754} C_VEL
LIN {X 0,Y 282.455,Z 1070.874,A -85,B 0,C 180,E1 4696.401,E2 4696.401} C_VEL
LIN {X 0,Y 294.008,Z 1050.81,A -85,B 0,C 180,E1 4695.263,E2 4695.263} C_VEL
LIN {X 0,Y 303.504,Z 1031.468,A -85,B 0,C 180,E1 4694.409,E2 4694.409} C_VEL
LIN {X 0,Y 312.785,Z 1009.099,A -85,B 0,C 180,E1 4693.646,E2 4693.646} C_VEL
LIN {X 0,Y 319.801,Z 988.481,A -85,B 0,C 180,E1 4693.119,E2 4693.119} C_VEL
LIN {X 0,Y 326.047,Z 964.951,A -85,B 0,C 180,E1 4692.664,E2 4692.664} C_VEL
LIN {X 0,Y 330.571,Z 941.537,A -85,B 0,C 180,E1 4692.286,E2 4692.286} C_VEL
LIN {X 0,Y 339.029,Z 868.099,A -85,B 0,C 180,E1 4691.304,E2 4691.304} C_VEL
LIN {X 0,Y 346.547,Z 800.776,A -85,B 0,C 180,E1 4690.389,E2 4690.389} C_VEL
LIN {X 0,Y 345.567,Z 796.21,A -85,B 0,C 180,E1 4687.983,E2 4687.983} C_VEL
LIN {X 0,Y 344.985,Z 793.095,A -85,B 0,C 180,E1 4685.489,E2 4685.489} C_VEL
LIN {X 0,Y 344.885,Z 791.646,A -85,B 0,C 180,E1 4683.823,E2 4683.823} C_VEL
LIN {X 0,Y 345.33,Z 790.971,A -85,B 0,C 180,E1 4680.332,E2 4680.332} C_VEL
LIN {X 0,Y 346.691,Z 792.73,A -85,B 0,C 180,E1 4677.024,E2 4677.024} C_VEL
LIN {X 0,Y 347.448,Z 794.648,A -85,B 0,C 180,E1 4675.657,E2 4675.657} C_VEL
LIN {X 0,Y 331.143,Z 935.579,A -85,B 0,C 180,E1 4673.72,E2 4673.72} C_VEL
LIN {X 0,Y 326.68,Z 959.475,A -85,B 0,C 180,E1 4673.307,E2 4673.307} C_VEL
LIN {X 0,Y 321.011,Z 981.848,A -85,B 0,C 180,E1 4672.808,E2 4672.808} C_VEL
LIN {X 0,Y 313.876,Z 1003.475,A -85,B 0,C 180,E1 4672.177,E2 4672.177} C_VEL
LIN {X 0,Y 311.038,Z 1011.266,A -85,B 0,C 180,E1 4671.906,E2 4671.906} C_VEL
LIN {X 0,Y 307.912,Z 1018.427,A -85,B 0,C 180,E1 4671.815,E2 4671.815} C_VEL
LIN {X 0,Y 298.869,Z 1036.299,A -85,B 0,C 180,E1 4672.195,E2 4672.195} C_VEL
LIN {X 0,Y 295.292,Z 1043.059,A -85,B 0,C 180,E1 4672.065,E2 4672.065} C_VEL
LIN {X 0,Y 284.463,Z 1062.815,A -85,B 0,C 180,E1 4670.997,E2 4670.997} C_VEL
LIN {X 0,Y 271.882,Z 1082.512,A -85,B 0,C 180,E1 4669.653,E2 4669.653} C_VEL
LIN {X 0,Y 258.557,Z 1100.961,A -85,B 0,C 180,E1 4668.061,E2 4668.061} C_VEL
LIN {X 0,Y 244.091,Z 1118.392,A -85,B 0,C 180,E1 4666.122,E2 4666.122} C_VEL
LIN {X 0,Y 228.192,Z 1135.504,A -85,B 0,C 180,E1 4663.654,E2 4663.654} C_VEL
LIN {X 0,Y 213.605,Z 1149.508,A -85,B 0,C 180,E1 4661.003,E2 4661.003} C_VEL
LIN {X 0,Y 196.416,Z 1164.354,A -85,B 0,C 180,E1 4657.239,E2 4657.239} C_VEL
LIN {X 0,Y 180.735,Z 1176.656,A -85,B 0,C 180,E1 4652.959,E2 4652.959} C_VEL
LIN {X 0,Y 165.589,Z 1187.404,A -85,B 0,C 180,E1 4647.709,E2 4647.709} C_VEL
LIN {X 0,Y 151.421,Z 1196.903,A -85,B 0,C 180,E1 4641.185,E2 4641.185} C_VEL
LIN {X 0,Y 139.419,Z 1204.481,A -85,B 0,C 180,E1 4633.509,E2 4633.509} C_VEL
LIN {X 0,Y 129.353,Z 1210.943,A -85,B 0,C 180,E1 4623.817,E2 4623.817} C_VEL
LIN {X 0,Y 123.53,Z 1215.015,A -85,B 0,C 180,E1 4614.381,E2 4614.381} C_VEL
LIN {X 0,Y 120.433,Z 1217.92,A -85,B 0,C 180,E1 4603.442,E2 4603.442} C_VEL
LIN {X 0,Y 119.984,Z 1218.981,A -85,B 0,C 180,E1 4594.78,E2 4594.78} C_VEL
LIN {X 0,Y 120.025,Z 1219.147,A -85,B 0,C 180,E1 4588.568,E2 4588.568} C_VEL
LIN {X 0,Y 120.053,Z 1218.559,A -85,B 0,C 180,E1 4580.895,E2 4580.895} C_VEL
LIN {X 0,Y 121.378,Z 1216.801,A -85,B 0,C 180,E1 4571.758,E2 4571.758} C_VEL
LIN {X 0,Y 125.668,Z 1213.453,A -85,B 0,C 180,E1 4561.486,E2 4561.486} C_VEL
LIN {X 0,Y 133.534,Z 1208.128,A -85,B 0,C 180,E1 4551.576,E2 4551.576} C_VEL
LIN {X 0,Y 144.568,Z 1201.17,A -85,B 0,C 180,E1 4542.852,E2 4542.852} C_VEL
LIN {X 0,Y 156.971,Z 1193.077,A -85,B 0,C 180,E1 4536.007,E2 4536.007} C_VEL
LIN {X 0,Y 171.9,Z 1182.88,A -85,B 0,C 180,E1 4529.927,E2 4529.927} C_VEL
LIN {X 0,Y 186.062,Z 1172.366,A -85,B 0,C 180,E1 4525.462,E2 4525.462} C_VEL
LIN {X 0,Y 202.777,Z 1158.835,A -85,B 0,C 180,E1 4521.264,E2 4521.264} C_VEL
LIN {X 0,Y 217.835,Z 1145.336,A -85,B 0,C 180,E1 4518.172,E2 4518.172} C_VEL
LIN {X 0,Y 233.433,Z 1129.768,A -85,B 0,C 180,E1 4515.478,E2 4515.478} C_VEL
LIN {X 0,Y 247.669,Z 1113.938,A -85,B 0,C 180,E1 4513.362,E2 4513.362} C_VEL
LIN {X 0,Y 262.2,Z 1095.635,A -85,B 0,C 180,E1 4511.47,E2 4511.47} C_VEL
LIN {X 0,Y 275.12,Z 1077.315,A -85,B 0,C 180,E1 4509.975,E2 4509.975} C_VEL
LIN {X 0,Y 287.264,Z 1057.325,A -85,B 0,C 180,E1 4508.699,E2 4508.699} C_VEL
LIN {X 0,Y 298.113,Z 1036.831,A -85,B 0,C 180,E1 4507.653,E2 4507.653} C_VEL
LIN {X 0,Y 307.138,Z 1016.579,A -85,B 0,C 180,E1 4506.833,E2 4506.833} C_VEL
LIN {X 0,Y 315.737,Z 993.462,A -85,B 0,C 180,E1 4506.09,E2 4506.09} C_VEL
LIN {X 0,Y 322.121,Z 971.946,A -85,B 0,C 180,E1 4505.553,E2 4505.553} C_VEL
LIN {X 0,Y 327.563,Z 947.651,A -85,B 0,C 180,E1 4505.097,E2 4505.097} C_VEL
LIN {X 0,Y 331.216,Z 924.001,A -85,B 0,C 180,E1 4504.752,E2 4504.752} C_VEL
LIN {X 0,Y 345.449,Z 800.656,A -85,B 0,C 180,E1 4503.111,E2 4503.111} C_VEL
LIN {X 0,Y 344.108,Z 798.547,A -85,B 0,C 180,E1 4499.833,E2 4499.833} C_VEL
LIN {X 0,Y 343.581,Z 798.993,A -85,B 0,C 180,E1 4496.83,E2 4496.83} C_VEL
LIN {X 0,Y 343.596,Z 800.036,A -85,B 0,C 180,E1 4495.159,E2 4495.159} C_VEL
LIN {X 0,Y 344.002,Z 803.169,A -85,B 0,C 180,E1 4492.568,E2 4492.568} C_VEL
LIN {X 0,Y 344.58,Z 806.204,A -85,B 0,C 180,E1 4490.816,E2 4490.816} C_VEL
LIN {X 0,Y 344.582,Z 806.703,A -85,B 0,C 180,E1 4490.718,E2 4490.718} C_VEL
LIN {X 0,Y 329.28,Z 939.521,A -85,B 0,C 180,E1 4489.018,E2 4489.018} C_VEL
LIN {X 0,Y 324.827,Z 963.08,A -85,B 0,C 180,E1 4488.66,E2 4488.66} C_VEL
LIN {X 0,Y 319.121,Z 985.221,A -85,B 0,C 180,E1 4488.269,E2 4488.269} C_VEL
LIN {X 0,Y 312.027,Z 1006.251,A -85,B 0,C 180,E1 4487.779,E2 4487.779} C_VEL
LIN {X 0,Y 303.108,Z 1028.217,A -85,B 0,C 180,E1 4487.099,E2 4487.099} C_VEL
LIN {X 0,Y 293.319,Z 1048.202,A -85,B 0,C 180,E1 4486.287,E2 4486.287} C_VEL
LIN {X 0,Y 280.909,Z 1069.83,A -85,B 0,C 180,E1 4485.15,E2 4485.15} C_VEL
LIN {X 0,Y 268.525,Z 1088.506,A -85,B 0,C 180,E1 4483.877,E2 4483.877} C_VEL
LIN {X 0,Y 255.009,Z 1106.177,A -85,B 0,C 180,E1 4482.321,E2 4482.321} C_VEL
LIN {X 0,Y 240.851,Z 1122.695,A -85,B 0,C 180,E1 4480.451,E2 4480.451} C_VEL
LIN {X 0,Y 225.283,Z 1138.584,A -85,B 0,C 180,E1 4478.062,E2 4478.062} C_VEL
LIN {X 0,Y 208.537,Z 1153.797,A -85,B 0,C 180,E1 4474.983,E2 4474.983} C_VEL
LIN {X 0,Y 193.292,Z 1166.206,A -85,B 0,C 180,E1 4471.566,E2 4471.566} C_VEL
LIN {X 0,Y 178.11,Z 1177.248,A -85,B 0,C 180,E1 4467.358,E2 4467.358} C_VEL
LIN {X 0,Y 163.394,Z 1187.114,A -85,B 0,C 180,E1 4462.128,E2 4462.128} C_VEL
LIN {X 0,Y 149.653,Z 1195.417,A -85,B 0,C 180,E1 4455.634,E2 4455.634} C_VEL
LIN {X 0,Y 137.633,Z 1202.343,A -85,B 0,C 180,E1 4447.606,E2 4447.606} C_VEL
LIN {X 0,Y 129.198,Z 1207.067,A -85,B 0,C 180,E1 4439.18,E2 4439.18} C_VEL
LIN {X 0,Y 122.963,Z 1210.753,A -85,B 0,C 180,E1 4428.489,E2 4428.489} C_VEL
LIN {X 0,Y 120.552,Z 1212.478,A -85,B 0,C 180,E1 4419.067,E2 4419.067} C_VEL
LIN {X 0,Y 120.075,Z 1213.078,A -85,B 0,C 180,E1 4410,E2 4410} C_VEL
LIN {X 0,Y 120.545,Z 1212.511,A -85,B 0,C 180,E1 4400.933,E2 4400.933} C_VEL
LIN {X 0,Y 122.931,Z 1210.809,A -85,B 0,C 180,E1 4391.506,E2 4391.506} C_VEL
LIN {X 0,Y 129.483,Z 1206.967,A -85,B 0,C 180,E1 4380.383,E2 4380.383} C_VEL
LIN {X 0,Y 138.975,Z 1201.721,A -85,B 0,C 180,E1 4371.25,E2 4371.25} C_VEL
LIN {X 0,Y 151.142,Z 1194.657,A -85,B 0,C 180,E1 4363.474,E2 4363.474} C_VEL
LIN {X 0,Y 165.309,Z 1185.983,A -85,B 0,C 180,E1 4357.023,E2 4357.023} C_VEL
LIN {X 0,Y 179.483,Z 1176.471,A -85,B 0,C 180,E1 4352.14,E2 4352.14} C_VEL
LIN {X 0,Y 195.549,Z 1164.616,A -85,B 0,C 180,E1 4347.803,E2 4347.803} C_VEL
LIN {X 0,Y 210.907,Z 1152.041,A -85,B 0,C 180,E1 4344.464,E2 4344.464} C_VEL
LIN {X 0,Y 226.038,Z 1138.128,A -85,B 0,C 180,E1 4341.734,E2 4341.734} C_VEL
LIN {X 0,Y 240.754,Z 1123.11,A -85,B 0,C 180,E1 4339.484,E2 4339.484} C_VEL
LIN {X 0,Y 254.915,Z 1106.668,A -85,B 0,C 180,E1 4337.613,E2 4337.613} C_VEL
LIN {X 0,Y 268.433,Z 1089.105,A -85,B 0,C 180,E1 4336.056,E2 4336.056} C_VEL
LIN {X 0,Y 280.76,Z 1070.581,A -85,B 0,C 180,E1 4334.788,E2 4334.788} C_VEL
LIN {X 0,Y 292.769,Z 1049.891,A -85,B 0,C 180,E1 4333.684,E2 4333.684} C_VEL
LIN {X 0,Y 302.554,Z 1030.098,A -85,B 0,C 180,E1 4332.866,E2 4332.866} C_VEL
LIN {X 0,Y 311.944,Z 1007.392,A -85,B 0,C 180,E1 4332.151,E2 4332.151} C_VEL
LIN {X 0,Y 319.275,Z 985.806,A -85,B 0,C 180,E1 4331.644,E2 4331.644} C_VEL
LIN {X 0,Y 325.25,Z 962.74,A -85,B 0,C 180,E1 4331.235,E2 4331.235} C_VEL
LIN {X 0,Y 329.76,Z 938.527,A -85,B 0,C 180,E1 4330.869,E2 4330.869} C_VEL
LIN {X 0,Y 344.972,Z 806.659,A -85,B 0,C 180,E1 4329.173,E2 4329.173} C_VEL
LIN {X 0,Y 344.365,Z 803.45,A -85,B 0,C 180,E1 4327.34,E2 4327.34} C_VEL
LIN {X 0,Y 343.93,Z 800.283,A -85,B 0,C 180,E1 4324.669,E2 4324.669} C_VEL
LIN {X 0,Y 343.916,Z 799.299,A -85,B 0,C 180,E1 4323,E2 4323} C_VEL
LIN {X 0,Y 344.5,Z 799.008,A -85,B 0,C 180,E1 4319.834,E2 4319.834} C_VEL
LIN {X 0,Y 345.742,Z 800.989,A -85,B 0,C 180,E1 4316.893,E2 4316.893} C_VEL
LIN {X 0,Y 329.929,Z 935.864,A -85,B 0,C 180,E1 4315.09,E2 4315.09} C_VEL
LIN {X 0,Y 325.404,Z 959.803,A -85,B 0,C 180,E1 4314.694,E2 4314.694} C_VEL
LIN {X 0,Y 319.583,Z 982.465,A -85,B 0,C 180,E1 4314.212,E2 4314.212} C_VEL
LIN {X 0,Y 312.393,Z 1003.911,A -85,B 0,C 180,E1 4313.615,E2 4313.615} C_VEL
LIN {X 0,Y 303.816,Z 1025.304,A -85,B 0,C 180,E1 4312.854,E2 4312.854} C_VEL
LIN {X 0,Y 295.292,Z 1043.059,A -85,B 0,C 180,E1 4312.065,E2 4312.065} C_VEL
LIN {X 0,Y 291.534,Z 1050.005,A -85,B 0,C 180,E1 4311.915,E2 4311.915} C_VEL
LIN {X 0,Y 280.707,Z 1066.876,A -85,B 0,C 180,E1 4312.164,E2 4312.164} C_VEL
LIN {X 0,Y 276.511,Z 1073.175,A -85,B 0,C 180,E1 4311.972,E2 4311.972} C_VEL
LIN {X 0,Y 262.569,Z 1093.208,A -85,B 0,C 180,E1 4310.493,E2 4310.493} C_VEL
LIN {X 0,Y 249.048,Z 1110.292,A -85,B 0,C 180,E1 4308.889,E2 4308.889} C_VEL
LIN {X 0,Y 234.083,Z 1126.952,A -85,B 0,C 180,E1 4306.874,E2 4306.874} C_VEL
LIN {X 0,Y 218.924,Z 1142.102,A -85,B 0,C 180,E1 4304.507,E2 4304.507} C_VEL
LIN {X 0,Y 202.475,Z 1156.661,A -85,B 0,C 180,E1 4301.465,E2 4301.465} C_VEL
LIN {X 0,Y 185.868,Z 1169.971,A -85,B 0,C 180,E1 4297.707,E2 4297.707} C_VEL
LIN {X 0,Y 170.174,Z 1181.222,A -85,B 0,C 180,E1 4293.262,E2 4293.262} C_VEL
LIN {X 0,Y 154.286,Z 1191.732,A -85,B 0,C 180,E1 4287.402,E2 4287.402} C_VEL
LIN {X 0,Y 140.82,Z 1199.967,A -85,B 0,C 180,E1 4280.708,E2 4280.708} C_VEL
LIN {X 0,Y 128.07,Z 1207.462,A -85,B 0,C 180,E1 4271.575,E2 4271.575} C_VEL
LIN {X 0,Y 119.431,Z 1212.672,A -85,B 0,C 180,E1 4261.831,E2 4261.831} C_VEL
LIN {X 0,Y 113.958,Z 1216.387,A -85,B 0,C 180,E1 4250.546,E2 4250.546} C_VEL
LIN {X 0,Y 112.158,Z 1218.228,A -85,B 0,C 180,E1 4240.79,E2 4240.79} C_VEL
LIN {X 0,Y 112.007,Z 1218.901,A -85,B 0,C 180,E1 4232.558,E2 4232.558} C_VEL
LIN {X 0,Y 111.997,Z 1218.845,A -85,B 0,C 180,E1 4226.417,E2 4226.417} C_VEL
LIN {X 0,Y 112.203,Z 1218.119,A -85,B 0,C 180,E1 4218.597,E2 4218.597} C_VEL
LIN {X 0,Y 114.282,Z 1216.11,A -85,B 0,C 180,E1 4208.441,E2 4208.441} C_VEL
LIN {X 0,Y 120.416,Z 1211.963,A -85,B 0,C 180,E1 4196.769,E2 4196.769} C_VEL
LIN {X 0,Y 129.495,Z 1206.585,A -85,B 0,C 180,E1 4187.184,E2 4187.184} C_VEL
LIN {X 0,Y 141.408,Z 1199.489,A -85,B 0,C 180,E1 4178.942,E2 4178.942} C_VEL
LIN {X 0,Y 155.654,Z 1190.773,A -85,B 0,C 180,E1 4172.014,E2 4172.014} C_VEL
LIN {X 0,Y 170.923,Z 1180.534,A -85,B 0,C 180,E1 4166.49,E2 4166.49} C_VEL
LIN {X 0,Y 187.169,Z 1168.788,A -85,B 0,C 180,E1 4161.96,E2 4161.96} C_VEL
LIN {X 0,Y 203.391,Z 1155.653,A -85,B 0,C 180,E1 4158.339,E2 4158.339} C_VEL
LIN {X 0,Y 220.674,Z 1140.101,A -85,B 0,C 180,E1 4155.185,E2 4155.185} C_VEL
LIN {X 0,Y 234.975,Z 1125.699,A -85,B 0,C 180,E1 4152.985,E2 4152.985} C_VEL
LIN {X 0,Y 250.497,Z 1108.129,A -85,B 0,C 180,E1 4150.916,E2 4150.916} C_VEL
LIN {X 0,Y 263.962,Z 1090.938,A -85,B 0,C 180,E1 4149.341,E2 4149.341} C_VEL
LIN {X 0,Y 277.125,Z 1071.681,A -85,B 0,C 180,E1 4147.952,E2 4147.952} C_VEL
LIN {X 0,Y 289.004,Z 1051.881,A -85,B 0,C 180,E1 4146.821,E2 4146.821} C_VEL
LIN {X 0,Y 299.533,Z 1031.086,A -85,B 0,C 180,E1 4145.88,E2 4145.88} C_VEL
LIN {X 0,Y 308.877,Z 1009.44,A -85,B 0,C 180,E1 4145.104,E2 4145.104} C_VEL
LIN {X 0,Y 316.015,Z 989.218,A -85,B 0,C 180,E1 4144.537,E2 4144.537} C_VEL
LIN {X 0,Y 322.568,Z 966.22,A -85,B 0,C 180,E1 4144.025,E2 4144.025} C_VEL
LIN {X 0,Y 327.253,Z 943.933,A -85,B 0,C 180,E1 4143.649,E2 4143.649} C_VEL
LIN {X 0,Y 331.448,Z 913.475,A -85,B 0,C 180,E1 4143.236,E2 4143.236} C_VEL
LIN {X 0,Y 343.848,Z 807.667,A -85,B 0,C 180,E1 4141.875,E2 4141.875} C_VEL
LIN {X 0,Y 342.999,Z 806.404,A -85,B 0,C 180,E1 4139.332,E2 4139.332} C_VEL
LIN {X 0,Y 342.607,Z 807.38,A -85,B 0,C 180,E1 4135.816,E2 4135.816} C_VEL
LIN {X 0,Y 342.936,Z 810.872,A -85,B 0,C 180,E1 4132.882,E2 4132.882} C_VEL
LIN {X 0,Y 343.169,Z 812.381,A -85,B 0,C 180,E1 4131.978,E2 4131.978} C_VEL
LIN {X 0,Y 328.279,Z 939.291,A -85,B 0,C 180,E1 4130.406,E2 4130.406} C_VEL
LIN {X 0,Y 323.774,Z 962.831,A -85,B 0,C 180,E1 4130.066,E2 4130.066} C_VEL
LIN {X 0,Y 317.838,Z 985.533,A -85,B 0,C 180,E1 4129.688,E2 4129.688} C_VEL
LIN {X 0,Y 310.44,Z 1007.112,A -85,B 0,C 180,E1 4129.214,E2 4129.214} C_VEL
LIN {X 0,Y 301.428,Z 1028.857,A -85,B 0,C 180,E1 4128.577,E2 4128.577} C_VEL
LIN {X 0,Y 291.53,Z 1048.764,A -85,B 0,C 180,E1 4127.812,E2 4127.812} C_VEL
LIN {X 0,Y 279.37,Z 1069.644,A -85,B 0,C 180,E1 4126.775,E2 4126.775} C_VEL
LIN {X 0,Y 266.87,Z 1088.25,A -85,B 0,C 180,E1 4125.58,E2 4125.58} C_VEL
LIN {X 0,Y 252.936,Z 1106.215,A -85,B 0,C 180,E1 4124.084,E2 4124.084} C_VEL
LIN {X 0,Y 238.278,Z 1122.988,A -85,B 0,C 180,E1 4122.275,E2 4122.275} C_VEL
LIN {X 0,Y 222.876,Z 1138.402,A -85,B 0,C 180,E1 4120.065,E2 4120.065} C_VEL
LIN {X 0,Y 205.729,Z 1153.657,A -85,B 0,C 180,E1 4117.119,E2 4117.119} C_VEL
LIN {X 0,Y 190.38,Z 1165.823,A -85,B 0,C 180,E1 4113.906,E2 4113.906} C_VEL
LIN {X 0,Y 173.777,Z 1177.541,A -85,B 0,C 180,E1 4109.579,E2 4109.579} C_VEL
LIN {X 0,Y 158.541,Z 1187.333,A -85,B 0,C 180,E1 4104.444,E2 4104.444} C_VEL
LIN {X 0,Y 144.093,Z 1195.634,A -85,B 0,C 180,E1 4097.942,E2 4097.942} C_VEL
LIN {X 0,Y 130.802,Z 1202.799,A -85,B 0,C 180,E1 4089.379,E2 4089.379} C_VEL
LIN {X 0,Y 121.465,Z 1207.678,A -85,B 0,C 180,E1 4080.141,E2 4080.141} C_VEL
LIN {X 0,Y 115.135,Z 1211.068,A -85,B 0,C 180,E1 4069.269,E2 4069.269} C_VEL
LIN {X 0,Y 112.557,Z 1212.748,A -85,B 0,C 180,E1 4059.201,E2 4059.201} C_VEL
LIN {X 0,Y 112.077,Z 1213.282,A -85,B 0,C 180,E1 4050,E2 4050} C_VEL
LIN {X 0,Y 112.63,Z 1212.706,A -85,B 0,C 180,E1 4040.206,E2 4040.206} C_VEL
LIN {X 0,Y 115.3,Z 1211.015,A -85,B 0,C 180,E1 4030.233,E2 4030.233} C_VEL
LIN {X 0,Y 122.501,Z 1207.175,A -85,B 0,C 180,E1 4018.509,E2 4018.509} C_VEL
LIN {X 0,Y 132.741,Z 1201.928,A -85,B 0,C 180,E1 4009.056,E2 4009.056} C_VEL
LIN {X 0,Y 145.287,Z 1195.083,A -85,B 0,C 180,E1 4001.353,E2 4001.353} C_VEL
LIN {X 0,Y 159.848,Z 1186.654,A -85,B 0,C 180,E1 3994.974,E2 3994.974} C_VEL
LIN {X 0,Y 174.539,Z 1177.199,A -85,B 0,C 180,E1 3990.116,E2 3990.116} C_VEL
LIN {X 0,Y 191.095,Z 1165.477,A -85,B 0,C 180,E1 3985.849,E2 3985.849} C_VEL
LIN {X 0,Y 205.998,Z 1153.667,A -85,B 0,C 180,E1 3982.75,E2 3982.75} C_VEL
LIN {X 0,Y 223.177,Z 1138.397,A -85,B 0,C 180,E1 3979.81,E2 3979.81} C_VEL
LIN {X 0,Y 238.19,Z 1123.395,A -85,B 0,C 180,E1 3977.658,E2 3977.658} C_VEL
LIN {X 0,Y 252.6,Z 1106.998,A -85,B 0,C 180,E1 3975.876,E2 3975.876} C_VEL
LIN {X 0,Y 266.328,Z 1089.49,A -85,B 0,C 180,E1 3974.398,E2 3974.398} C_VEL
LIN {X 0,Y 278.825,Z 1071.017,A -85,B 0,C 180,E1 3973.197,E2 3973.197} C_VEL
LIN {X 0,Y 290.515,Z 1051.335,A -85,B 0,C 180,E1 3972.195,E2 3972.195} C_VEL
LIN {X 0,Y 300.405,Z 1031.724,A -85,B 0,C 180,E1 3971.421,E2 3971.421} C_VEL
LIN {X 0,Y 309.891,Z 1009.511,A -85,B 0,C 180,E1 3970.747,E2 3970.747} C_VEL
LIN {X 0,Y 317.048,Z 989.028,A -85,B 0,C 180,E1 3970.283,E2 3970.283} C_VEL
LIN {X 0,Y 323.657,Z 964.879,A -85,B 0,C 180,E1 3969.868,E2 3969.868} C_VEL
LIN {X 0,Y 328.324,Z 941.496,A -85,B 0,C 180,E1 3969.526,E2 3969.526} C_VEL
LIN {X 0,Y 336.473,Z 873.658,A -85,B 0,C 180,E1 3968.675,E2 3968.675} C_VEL
LIN {X 0,Y 343.528,Z 812.459,A -85,B 0,C 180,E1 3967.906,E2 3967.906} C_VEL
LIN {X 0,Y 342.993,Z 809.059,A -85,B 0,C 180,E1 3965.353,E2 3965.353} C_VEL
LIN {X 0,Y 342.928,Z 807.44,A -85,B 0,C 180,E1 3963.51,E2 3963.51} C_VEL
LIN {X 0,Y 343.426,Z 806.88,A -85,B 0,C 180,E1 3960.167,E2 3960.167} C_VEL
LIN {X 0,Y 344.115,Z 808.113,A -85,B 0,C 180,E1 3958.124,E2 3958.124} C_VEL
LIN {X 0,Y 328.905,Z 936.15,A -85,B 0,C 180,E1 3956.47,E2 3956.47} C_VEL
LIN {X 0,Y 324.341,Z 960.037,A -85,B 0,C 180,E1 3956.094,E2 3956.094} C_VEL
LIN {X 0,Y 318.621,Z 982.107,A -85,B 0,C 180,E1 3955.651,E2 3955.651} C_VEL
LIN {X 0,Y 311.108,Z 1004.349,A -85,B 0,C 180,E1 3955.066,E2 3955.066} C_VEL
LIN {X 0,Y 302.126,Z 1026.318,A -85,B 0,C 180,E1 3954.321,E2 3954.321} C_VEL
LIN {X 0,Y 291.877,Z 1047.066,A -85,B 0,C 180,E1 3953.427,E2 3953.427} C_VEL
LIN {X 0,Y 279.502,Z 1068.472,A -85,B 0,C 180,E1 3952.266,E2 3952.266} C_VEL
LIN {X 0,Y 276.511,Z 1073.175,A -85,B 0,C 180,E1 3951.972,E2 3951.972} C_VEL
LIN {X 0,Y 272.177,Z 1079.561,A -85,B 0,C 180,E1 3951.758,E2 3951.758} C_VEL
LIN {X 0,Y 259.735,Z 1095.37,A -85,B 0,C 180,E1 3951.862,E2 3951.862} C_VEL
LIN {X 0,Y 254.846,Z 1101.254,A -85,B 0,C 180,E1 3951.579,E2 3951.579} C_VEL
LIN {X 0,Y 239.741,Z 1118.783,A -85,B 0,C 180,E1 3949.818,E2 3949.818} C_VEL
LIN {X 0,Y 223.194,Z 1135.806,A -85,B 0,C 180,E1 3947.577,E2 3947.577} C_VEL
LIN {X 0,Y 207.031,Z 1150.543,A -85,B 0,C 180,E1 3944.994,E2 3944.994} C_VEL
LIN {X 0,Y 189.635,Z 1164.606,A -85,B 0,C 180,E1 3941.632,E2 3941.632} C_VEL
LIN {X 0,Y 172.669,Z 1176.992,A -85,B 0,C 180,E1 3937.53,E2 3937.53} C_VEL
LIN {X 0,Y 156.59,Z 1187.422,A -85,B 0,C 180,E1 3932.565,E2 3932.565} C_VEL
LIN {X 0,Y 140.933,Z 1196.834,A -85,B 0,C 180,E1 3926.105,E2 3926.105} C_VEL
LIN {X 0,Y 127.342,Z 1204.365,A -85,B 0,C 180,E1 3918.238,E2 3918.238} C_VEL
LIN {X 0,Y 115.586,Z 1210.735,A -85,B 0,C 180,E1 3907.892,E2 3907.892} C_VEL
LIN {X 0,Y 108.535,Z 1214.761,A -85,B 0,C 180,E1 3897.427,E2 3897.427} C_VEL
LIN {X 0,Y 104.611,Z 1217.58,A -85,B 0,C 180,E1 3884.955,E2 3884.955} C_VEL
LIN {X 0,Y 103.987,Z 1218.572,A -85,B 0,C 180,E1 3875.518,E2 3875.518} C_VEL
LIN {X 0,Y 104.023,Z 1218.738,A -85,B 0,C 180,E1 3868.348,E2 3868.348} C_VEL
LIN {X 0,Y 104.135,Z 1218.146,A -85,B 0,C 180,E1 3859.489,E2 3859.489} C_VEL
LIN {X 0,Y 105.997,Z 1216.384,A -85,B 0,C 180,E1 3848.995,E2 3848.995} C_VEL
LIN {X 0,Y 111.484,Z 1213.031,A -85,B 0,C 180,E1 3837.444,E2 3837.444} C_VEL
LIN {X 0,Y 120.516,Z 1207.961,A -85,B 0,C 180,E1 3827.132,E2 3827.132} C_VEL
LIN {X 0,Y 132.607,Z 1201.443,A -85,B 0,C 180,E1 3818.357,E2 3818.357} C_VEL
LIN {X 0,Y 147.112,Z 1193.046,A -85,B 0,C 180,E1 3811.089,E2 3811.089} C_VEL
LIN {X 0,Y 163.463,Z 1182.936,A -85,B 0,C 180,E1 3805.14,E2 3805.14} C_VEL
LIN {X 0,Y 179.54,Z 1171.893,A -85,B 0,C 180,E1 3800.677,E2 3800.677} C_VEL
LIN {X 0,Y 197.374,Z 1158.314,A -85,B 0,C 180,E1 3796.777,E2 3796.777} C_VEL
LIN {X 0,Y 213.258,Z 1144.795,A -85,B 0,C 180,E1 3793.948,E2 3793.948} C_VEL
LIN {X 0,Y 229.581,Z 1129.158,A -85,B 0,C 180,E1 3791.506,E2 3791.506} C_VEL
LIN {X 0,Y 244.86,Z 1112.779,A -85,B 0,C 180,E1 3789.551,E2 3789.551} C_VEL
LIN {X 0,Y 259.434,Z 1094.877,A -85,B 0,C 180,E1 3787.915,E2 3787.915} C_VEL
LIN {X 0,Y 273.238,Z 1075.689,A -85,B 0,C 180,E1 3786.537,E2 3786.537} C_VEL
LIN {X 0,Y 285.249,Z 1056.304,A -85,B 0,C 180,E1 3785.45,E2 3785.45} C_VEL
LIN {X 0,Y 296.864,Z 1034.502,A -85,B 0,C 180,E1 3784.48,E2 3784.48} C_VEL
LIN {X 0,Y 305.974,Z 1014.257,A -85,B 0,C 180,E1 3783.769,E2 3783.769} C_VEL
LIN {X 0,Y 314.181,Z 992.127,A -85,B 0,C 180,E1 3783.156,E2 3783.156} C_VEL
LIN {X 0,Y 320.691,Z 970.355,A -85,B 0,C 180,E1 3782.679,E2 3782.679} C_VEL
LIN {X 0,Y 325.881,Z 946.987,A -85,B 0,C 180,E1 3782.293,E2 3782.293} C_VEL
LIN {X 0,Y 329.616,Z 922.571,A -85,B 0,C 180,E1 3781.97,E2 3781.97} C_VEL
LIN {X 0,Y 342.384,Z 814.806,A -85,B 0,C 180,E1 3780.627,E2 3780.627} C_VEL
LIN {X 0,Y 341.828,Z 814.403,A -85,B 0,C 180,E1 3778.491,E2 3778.491} C_VEL
LIN {X 0,Y 341.611,Z 815.468,A -85,B 0,C 180,E1 3775.804,E2 3775.804} C_VEL
LIN {X 0,Y 341.859,Z 818.508,A -85,B 0,C 180,E1 3773.244,E2 3773.244} C_VEL
LIN {X 0,Y 327.472,Z 939.061,A -85,B 0,C 180,E1 3771.802,E2 3771.802} C_VEL
LIN {X 0,Y 322.924,Z 962.56,A -85,B 0,C 180,E1 3771.48,E2 3771.48} C_VEL
LIN {X 0,Y 316.994,Z 985.084,A -85,B 0,C 180,E1 3771.132,E2 3771.132} C_VEL
LIN {X 0,Y 309.313,Z 1007.271,A -85,B 0,C 180,E1 3770.681,E2 3770.681} C_VEL
LIN {X 0,Y 299.95,Z 1029.497,A -85,B 0,C 180,E1 3770.07,E2 3770.07} C_VEL
LIN {X 0,Y 289.95,Z 1049.325,A -85,B 0,C 180,E1 3769.354,E2 3769.354} C_VEL
LIN {X 0,Y 277.649,Z 1070.09,A -85,B 0,C 180,E1 3768.382,E2 3768.382} C_VEL
LIN {X 0,Y 264.522,Z 1089.311,A -85,B 0,C 180,E1 3767.214,E2 3767.214} C_VEL
LIN {X 0,Y 250.138,Z 1107.407,A -85,B 0,C 180,E1 3765.772,E2 3765.772} C_VEL
LIN {X 0,Y 235.044,Z 1124.199,A -85,B 0,C 180,E1 3764.026,E2 3764.026} C_VEL
LIN {X 0,Y 219.767,Z 1139.141,A -85,B 0,C 180,E1 3761.965,E2 3761.965} C_VEL
LIN {X 0,Y 202.233,Z 1154.303,A -85,B 0,C 180,E1 3759.137,E2 3759.137} C_VEL
LIN {X 0,Y 185.301,Z 1167.312,A -85,B 0,C 180,E1 3755.769,E2 3755.769} C_VEL
LIN {X 0,Y 169.129,Z 1178.213,A -85,B 0,C 180,E1 3751.746,E2 3751.746} C_VEL
LIN {X 0,Y 152.511,Z 1188.347,A -85,B 0,C 180,E1 3746.368,E2 3746.368} C_VEL
LIN {X 0,Y 138.141,Z 1196.196,A -85,B 0,C 180,E1 3740.105,E2 3740.105} C_VEL
LIN {X 0,Y 124.111,Z 1203.257,A -85,B 0,C 180,E1 3731.346,E2 3731.346} C_VEL
LIN {X 0,Y 113.77,Z 1208.289,A -85,B 0,C 180,E1 3721.233,E2 3721.233} C_VEL
LIN {X 0,Y 107.125,Z 1211.492,A -85,B 0,C 180,E1 3709.634,E2 3709.634} C_VEL
LIN {X 0,Y 104.437,Z 1213.149,A -85,B 0,C 180,E1 3698.257,E2 3698.257} C_VEL
LIN {X 0,Y 104.076,Z 1213.455,A -85,B 0,C 180,E1 3688.899,E2 3688.899} C_VEL
LIN {X 0,Y 104.79,Z 1212.857,A -85,B 0,C 180,E1 3678.999,E2 3678.999} C_VEL
LIN {X 0,Y 107.962,Z 1211.112,A -85,B 0,C 180,E1 3668.257,E2 3668.257} C_VEL
LIN {X 0,Y 115.665,Z 1207.383,A -85,B 0,C 180,E1 3656.41,E2 3656.41} C_VEL
LIN {X 0,Y 126.72,Z 1202.136,A -85,B 0,C 180,E1 3646.65,E2 3646.65} C_VEL
LIN {X 0,Y 140.004,Z 1195.32,A -85,B 0,C 180,E1 3638.883,E2 3638.883} C_VEL
LIN {X 0,Y 155.338,Z 1186.872,A -85,B 0,C 180,E1 3632.52,E2 3632.52} C_VEL
LIN {X 0,Y 170.617,Z 1177.42,A -85,B 0,C 180,E1 3627.761,E2 3627.761} C_VEL
LIN {X 0,Y 187.706,Z 1165.713,A -85,B 0,C 180,E1 3623.624,E2 3623.624} C_VEL
LIN {X 0,Y 203.01,Z 1153.911,A -85,B 0,C 180,E1 3620.645,E2 3620.645} C_VEL
LIN {X 0,Y 220.574,Z 1138.666,A -85,B 0,C 180,E1 3617.838,E2 3617.838} C_VEL
LIN {X 0,Y 235.873,Z 1123.681,A -85,B 0,C 180,E1 3615.794,E2 3615.794} C_VEL
LIN {X 0,Y 250.87,Z 1106.912,A -85,B 0,C 180,E1 3614.071,E2 3614.071} C_VEL
LIN {X 0,Y 264.915,Z 1089.234,A -85,B 0,C 180,E1 3612.672,E2 3612.672} C_VEL
LIN {X 0,Y 277.579,Z 1070.724,A -85,B 0,C 180,E1 3611.547,E2 3611.547} C_VEL
LIN {X 0,Y 289.408,Z 1050.992,A -85,B 0,C 180,E1 3610.611,E2 3610.611} C_VEL
LIN {X 0,Y 299.406,Z 1031.353,A -85,B 0,C 180,E1 3609.889,E2 3609.889} C_VEL
LIN {X 0,Y 308.985,Z 1009.079,A -85,B 0,C 180,E1 3609.263,E2 3609.263} C_VEL
LIN {X 0,Y 316.207,Z 988.564,A -85,B 0,C 180,E1 3608.835,E2 3608.835} C_VEL
LIN {X 0,Y 322.832,Z 964.499,A -85,B 0,C 180,E1 3608.451,E2 3608.451} C_VEL
LIN {X 0,Y 327.555,Z 941.024,A -85,B 0,C 180,E1 3608.127,E2 3608.127} C_VEL
LIN {X 0,Y 336.099,Z 870.837,A -85,B 0,C 180,E1 3607.28,E2 3607.28} C_VEL
LIN {X 0,Y 342.194,Z 818.736,A -85,B 0,C 180,E1 3606.628,E2 3606.628} C_VEL
LIN {X 0,Y 341.955,Z 815.462,A -85,B 0,C 180,E1 3603.688,E2 3603.688} C_VEL
LIN {X 0,Y 342.405,Z 814.796,A -85,B 0,C 180,E1 3600.335,E2 3600.335} C_VEL
LIN {X 0,Y 342.658,Z 815.382,A -85,B 0,C 180,E1 3599.368,E2 3599.368} C_VEL
LIN {X 0,Y 328.042,Z 936.652,A -85,B 0,C 180,E1 3597.854,E2 3597.854} C_VEL
LIN {X 0,Y 323.433,Z 960.444,A -85,B 0,C 180,E1 3597.498,E2 3597.498} C_VEL
LIN {X 0,Y 317.641,Z 982.534,A -85,B 0,C 180,E1 3597.08,E2 3597.08} C_VEL
LIN {X 0,Y 310.024,Z 1004.788,A -85,B 0,C 180,E1 3596.527,E2 3596.527} C_VEL
LIN {X 0,Y 300.76,Z 1027.073,A -85,B 0,C 180,E1 3595.812,E2 3595.812} C_VEL
LIN {X 0,Y 291.055,Z 1046.503,A -85,B 0,C 180,E1 3595.025,E2 3595.025} C_VEL
LIN {X 0,Y 278.999,Z 1067.281,A -85,B 0,C 180,E1 3593.979,E2 3593.979} C_VEL
LIN {X 0,Y 267.038,Z 1085.079,A -85,B 0,C 180,E1 3592.851,E2 3592.851} C_VEL
LIN {X 0,Y 254.846,Z 1101.254,A -85,B 0,C 180,E1 3591.579,E2 3591.579} C_VEL
LIN {X 0,Y 249.824,Z 1107.05,A -85,B 0,C 180,E1 3591.271,E2 3591.271} C_VEL
LIN {X 0,Y 235.064,Z 1122.29,A -85,B 0,C 180,E1 3591.168,E2 3591.168} C_VEL
LIN {X 0,Y 230.435,Z 1126.819,A -85,B 0,C 180,E1 3590.807,E2 3590.807} C_VEL
LIN {X 0,Y 214.18,Z 1142.396,A -85,B 0,C 180,E1 3588.62,E2 3588.62} C_VEL
LIN {X 0,Y 196.939,Z 1156.867,A -85,B 0,C 180,E1 3585.861,E2 3585.861} C_VEL
LIN {X 0,Y 179.368,Z 1170.086,A -85,B 0,C 180,E1 3582.404,E2 3582.404} C_VEL
LIN {X 0,Y 162.558,Z 1181.287,A -85,B 0,C 180,E1 3578.243,E2 3578.243} C_VEL
LIN {X 0,Y 144.5,Z 1192.122,A -85,B 0,C 180,E1 3572.336,E2 3572.336} C_VEL
LIN {X 0,Y 129.602,Z 1200.255,A -85,B 0,C 180,E1 3565.638,E2 3565.638} C_VEL
LIN {X 0,Y 115.664,Z 1207.302,A -85,B 0,C 180,E1 3556.564,E2 3556.564} C_VEL
LIN {X 0,Y 105.398,Z 1212.464,A -85,B 0,C 180,E1 3546.027,E2 3546.027} C_VEL
LIN {X 0,Y 98.607,Z 1216.09,A -85,B 0,C 180,E1 3533.294,E2 3533.294} C_VEL
LIN {X 0,Y 96.237,Z 1217.887,A -85,B 0,C 180,E1 3521.993,E2 3521.993} C_VEL
LIN {X 0,Y 96.012,Z 1218.516,A -85,B 0,C 180,E1 3512.387,E2 3512.387} C_VEL
LIN {X 0,Y 95.99,Z 1218.41,A -85,B 0,C 180,E1 3505.22,E2 3505.22} C_VEL
LIN {X 0,Y 96.501,Z 1217.572,A -85,B 0,C 180,E1 3495.601,E2 3495.601} C_VEL
LIN {X 0,Y 100.274,Z 1215.134,A -85,B 0,C 180,E1 3482.558,E2 3482.558} C_VEL
LIN {X 0,Y 107.855,Z 1211.104,A -85,B 0,C 180,E1 3470.921,E2 3470.921} C_VEL
LIN {X 0,Y 119.598,Z 1205.303,A -85,B 0,C 180,E1 3460.468,E2 3460.468} C_VEL
LIN {X 0,Y 133.668,Z 1197.957,A -85,B 0,C 180,E1 3452.301,E2 3452.301} C_VEL
LIN {X 0,Y 150.593,Z 1188.46,A -85,B 0,C 180,E1 3445.449,E2 3445.449} C_VEL
LIN {X 0,Y 166.673,Z 1178.486,A -85,B 0,C 180,E1 3440.637,E2 3440.637} C_VEL
LIN {X 0,Y 184.556,Z 1166.091,A -85,B 0,C 180,E1 3436.48,E2 3436.48} C_VEL
LIN {X 0,Y 201.42,Z 1153.061,A -85,B 0,C 180,E1 3433.357,E2 3433.357} C_VEL
LIN {X 0,Y 217.853,Z 1138.669,A -85,B 0,C 180,E1 3430.836,E2 3430.836} C_VEL
LIN {X 0,Y 234.176,Z 1122.735,A -85,B 0,C 180,E1 3428.724,E2 3428.724} C_VEL
LIN {X 0,Y 249.562,Z 1105.476,A -85,B 0,C 180,E1 3427.002,E2 3427.002} C_VEL
LIN {X 0,Y 264.206,Z 1086.902,A -85,B 0,C 180,E1 3425.563,E2 3425.563} C_VEL
LIN {X 0,Y 276.795,Z 1068.533,A -85,B 0,C 180,E1 3424.452,E2 3424.452} C_VEL
LIN {X 0,Y 289.477,Z 1047.114,A -85,B 0,C 180,E1 3423.429,E2 3423.429} C_VEL
LIN {X 0,Y 299.73,Z 1026.827,A -85,B 0,C 180,E1 3422.66,E2 3422.66} C_VEL
LIN {X 0,Y 308.869,Z 1005.006,A -85,B 0,C 180,E1 3422.004,E2 3422.004} C_VEL
LIN {X 0,Y 316.622,Z 982.529,A -85,B 0,C 180,E1 3421.481,E2 3421.481} C_VEL
LIN {X 0,Y 322.547,Z 960.047,A -85,B 0,C 180,E1 3421.082,E2 3421.082} C_VEL
LIN {X 0,Y 327.277,Z 935.289,A -85,B 0,C 180,E1 3420.737,E2 3420.737} C_VEL
LIN {X 0,Y 341.032,Z 822.289,A -85,B 0,C 180,E1 3419.355,E2 3419.355} C_VEL
LIN {X 0,Y 340.629,Z 823.183,A -85,B 0,C 180,E1 3416.129,E2 3416.129} C_VEL
LIN {X 0,Y 340.655,Z 825.14,A -85,B 0,C 180,E1 3414.51,E2 3414.51} C_VEL
LIN {X 0,Y 326.859,Z 938.831,A -85,B 0,C 180,E1 3413.203,E2 3413.203} C_VEL
LIN {X 0,Y 322.237,Z 962.431,A -85,B 0,C 180,E1 3412.9,E2 3412.9} C_VEL
LIN {X 0,Y 316.108,Z 985.38,A -85,B 0,C 180,E1 3412.571,E2 3412.571} C_VEL
LIN {X 0,Y 308.826,Z 1006.285,A -85,B 0,C 180,E1 3412.182,E2 3412.182} C_VEL
LIN {X 0,Y 299.644,Z 1028.141,A -85,B 0,C 180,E1 3411.636,E2 3411.636} C_VEL
LIN {X 0,Y 289.541,Z 1048.1,A -85,B 0,C 180,E1 3410.977,E2 3410.977} C_VEL
LIN {X 0,Y 276.626,Z 1069.807,A -85,B 0,C 180,E1 3410.044,E2 3410.044} C_VEL
LIN {X 0,Y 263.81,Z 1088.398,A -85,B 0,C 180,E1 3409,E2 3409} C_VEL
LIN {X 0,Y 249.691,Z 1106.096,A -85,B 0,C 180,E1 3407.706,E2 3407.706} C_VEL
LIN {X 0,Y 234.806,Z 1122.651,A -85,B 0,C 180,E1 3406.137,E2 3406.137} C_VEL
LIN {X 0,Y 218.313,Z 1138.585,A -85,B 0,C 180,E1 3404.109,E2 3404.109} C_VEL
LIN {X 0,Y 200.381,Z 1153.861,A -85,B 0,C 180,E1 3401.452,E2 3401.452} C_VEL
LIN {X 0,Y 183.836,Z 1166.31,A -85,B 0,C 180,E1 3398.442,E2 3398.442} C_VEL
LIN {X 0,Y 166.261,Z 1177.935,A -85,B 0,C 180,E1 3394.431,E2 3394.431} C_VEL
LIN {X 0,Y 149.557,Z 1187.834,A -85,B 0,C 180,E1 3389.462,E2 3389.462} C_VEL
LIN {X 0,Y 133.761,Z 1196.066,A -85,B 0,C 180,E1 3383.113,E2 3383.113} C_VEL
LIN {X 0,Y 118.342,Z 1203.38,A -85,B 0,C 180,E1 3374.095,E2 3374.095} C_VEL
LIN {X 0,Y 107.338,Z 1208.298,A -85,B 0,C 180,E1 3363.98,E2 3363.98} C_VEL
LIN {X 0,Y 99.788,Z 1211.591,A -85,B 0,C 180,E1 3351.761,E2 3351.761} C_VEL
LIN {X 0,Y 96.569,Z 1213.29,A -85,B 0,C 180,E1 3339.536,E2 3339.536} C_VEL
LIN {X 0,Y 96.078,Z 1213.681,A -85,B 0,C 180,E1 3329.404,E2 3329.404} C_VEL
LIN {X 0,Y 96.909,Z 1213.062,A -85,B 0,C 180,E1 3318.092,E2 3318.092} C_VEL
LIN {X 0,Y 100.502,Z 1211.317,A -85,B 0,C 180,E1 3306.55,E2 3306.55} C_VEL
LIN {X 0,Y 109.003,Z 1207.59,A -85,B 0,C 180,E1 3294.052,E2 3294.052} C_VEL
LIN {X 0,Y 120.359,Z 1202.591,A -85,B 0,C 180,E1 3284.404,E2 3284.404} C_VEL
LIN {X 0,Y 134.366,Z 1195.876,A -85,B 0,C 180,E1 3276.519,E2 3276.519} C_VEL
LIN {X 0,Y 150.366,Z 1187.539,A -85,B 0,C 180,E1 3270.182,E2 3270.182} C_VEL
LIN {X 0,Y 166.995,Z 1177.642,A -85,B 0,C 180,E1 3265.3,E2 3265.3} C_VEL
LIN {X 0,Y 184.611,Z 1165.953,A -85,B 0,C 180,E1 3261.322,E2 3261.322} C_VEL
LIN {X 0,Y 200.303,Z 1154.155,A -85,B 0,C 180,E1 3258.482,E2 3258.482} C_VEL
LIN {X 0,Y 218.239,Z 1138.94,A -85,B 0,C 180,E1 3255.823,E2 3255.823} C_VEL
LIN {X 0,Y 232.886,Z 1124.882,A -85,B 0,C 180,E1 3254.001,E2 3254.001} C_VEL
LIN {X 0,Y 248.883,Z 1107.43,A -85,B 0,C 180,E1 3252.294,E2 3252.294} C_VEL
LIN {X 0,Y 263.273,Z 1089.611,A -85,B 0,C 180,E1 3250.97,E2 3250.97} C_VEL
LIN {X 0,Y 276.089,Z 1071.162,A -85,B 0,C 180,E1 3249.92,E2 3249.92} C_VEL
LIN {X 0,Y 288.044,Z 1051.542,A -85,B 0,C 180,E1 3249.05,E2 3249.05} C_VEL
LIN {X 0,Y 298.502,Z 1031.23,A -85,B 0,C 180,E1 3248.357,E2 3248.357} C_VEL
LIN {X 0,Y 308.288,Z 1008.647,A -85,B 0,C 180,E1 3247.772,E2 3247.772} C_VEL
LIN {X 0,Y 315.569,Z 988.1,A -85,B 0,C 180,E1 3247.38,E2 3247.38} C_VEL
LIN {X 0,Y 322.178,Z 964.236,A -85,B 0,C 180,E1 3247.03,E2 3247.03} C_VEL
LIN {X 0,Y 326.953,Z 940.75,A -85,B 0,C 180,E1 3246.725,E2 3246.725} C_VEL
LIN {X 0,Y 335.233,Z 873.773,A -85,B 0,C 180,E1 3245.949,E2 3245.949} C_VEL
LIN {X 0,Y 341.022,Z 825.185,A -85,B 0,C 180,E1 3245.384,E2 3245.384} C_VEL
LIN {X 0,Y 340.983,Z 823.234,A -85,B 0,C 180,E1 3243.194,E2 3243.194} C_VEL
LIN {X 0,Y 341.341,Z 822.842,A -85,B 0,C 180,E1 3240.621,E2 3240.621} C_VEL
LIN {X 0,Y 327.372,Z 937.154,A -85,B 0,C 180,E1 3239.245,E2 3239.245} C_VEL
LIN {X 0,Y 322.73,Z 960.806,A -85,B 0,C 180,E1 3238.911,E2 3238.911} C_VEL
LIN {X 0,Y 316.811,Z 983.129,A -85,B 0,C 180,E1 3238.513,E2 3238.513} C_VEL
LIN {X 0,Y 309.144,Z 1005.226,A -85,B 0,C 180,E1 3237.998,E2 3237.998} C_VEL
LIN {X 0,Y 300.274,Z 1026.432,A -85,B 0,C 180,E1 3237.363,E2 3237.363} C_VEL
LIN {X 0,Y 289.971,Z 1046.851,A -85,B 0,C 180,E1 3236.593,E2 3236.593} C_VEL
LIN {X 0,Y 277.773,Z 1067.578,A -85,B 0,C 180,E1 3235.614,E2 3235.614} C_VEL
LIN {X 0,Y 265.658,Z 1085.351,A -85,B 0,C 180,E1 3234.559,E2 3234.559} C_VEL
LIN {X 0,Y 250.297,Z 1105.008,A -85,B 0,C 180,E1 3233.061,E2 3233.061} C_VEL
LIN {X 0,Y 235.124,Z 1122.064,A -85,B 0,C 180,E1 3231.377,E2 3231.377} C_VEL
LIN {X 0,Y 230.435,Z 1126.819,A -85,B 0,C 180,E1 3230.807,E2 3230.807} C_VEL
LIN {X 0,Y 224.927,Z 1132.169,A -85,B 0,C 180,E1 3230.383,E2 3230.383} C_VEL
LIN {X 0,Y 209.524,Z 1145.031,A -85,B 0,C 180,E1 3230.073,E2 3230.073} C_VEL
LIN {X 0,Y 203.719,Z 1149.718,A -85,B 0,C 180,E1 3229.551,E2 3229.551} C_VEL
LIN {X 0,Y 185.081,Z 1164.118,A -85,B 0,C 180,E1 3226.509,E2 3226.509} C_VEL
LIN {X 0,Y 167.388,Z 1176.285,A -85,B 0,C 180,E1 3222.887,E2 3222.887} C_VEL
LIN {X 0,Y 149.666,Z 1186.974,A -85,B 0,C 180,E1 3218.218,E2 3218.218} C_VEL
LIN {X 0,Y 132.365,Z 1196.412,A -85,B 0,C 180,E1 3212.073,E2 3212.073} C_VEL
LIN {X 0,Y 116.955,Z 1203.931,A -85,B 0,C 180,E1 3204.307,E2 3204.307} C_VEL
LIN {X 0,Y 102.553,Z 1210.529,A -85,B 0,C 180,E1 3193.037,E2 3193.037} C_VEL
LIN {X 0,Y 93.935,Z 1214.508,A -85,B 0,C 180,E1 3181.437,E2 3181.437} C_VEL
LIN {X 0,Y 88.876,Z 1217.24,A -85,B 0,C 180,E1 3167.004,E2 3167.004} C_VEL
LIN {X 0,Y 87.994,Z 1218.187,A -85,B 0,C 180,E1 3155.87,E2 3155.87} C_VEL
LIN {X 0,Y 88.02,Z 1218.329,A -85,B 0,C 180,E1 3148.047,E2 3148.047} C_VEL
LIN {X 0,Y 88.21,Z 1217.804,A -85,B 0,C 180,E1 3138.227,E2 3138.227} C_VEL
LIN {X 0,Y 90.701,Z 1216.084,A -85,B 0,C 180,E1 3125.929,E2 3125.929} C_VEL
LIN {X 0,Y 97.588,Z 1212.779,A -85,B 0,C 180,E1 3112.807,E2 3112.807} C_VEL
LIN {X 0,Y 108.968,Z 1207.532,A -85,B 0,C 180,E1 3101.201,E2 3101.201} C_VEL
LIN {X 0,Y 122.997,Z 1201.005,A -85,B 0,C 180,E1 3092.283,E2 3092.283} C_VEL
LIN {X 0,Y 139.262,Z 1192.598,A -85,B 0,C 180,E1 3085.225,E2 3085.225} C_VEL
LIN {X 0,Y 157.126,Z 1182.464,A -85,B 0,C 180,E1 3079.647,E2 3079.647} C_VEL
LIN {X 0,Y 173.821,Z 1171.781,A -85,B 0,C 180,E1 3075.686,E2 3075.686} C_VEL
LIN {X 0,Y 193.244,Z 1157.795,A -85,B 0,C 180,E1 3072.069,E2 3072.069} C_VEL
LIN {X 0,Y 209.888,Z 1144.258,A -85,B 0,C 180,E1 3069.565,E2 3069.565} C_VEL
LIN {X 0,Y 226.868,Z 1128.556,A -85,B 0,C 180,E1 3067.421,E2 3067.421} C_VEL
LIN {X 0,Y 242.673,Z 1112.132,A -85,B 0,C 180,E1 3065.719,E2 3065.719} C_VEL
LIN {X 0,Y 257.322,Z 1094.587,A -85,B 0,C 180,E1 3064.331,E2 3064.331} C_VEL
LIN {X 0,Y 271.37,Z 1075.516,A -85,B 0,C 180,E1 3063.145,E2 3063.145} C_VEL
LIN {X 0,Y 283.372,Z 1056.599,A -85,B 0,C 180,E1 3062.224,E2 3062.224} C_VEL
LIN {X 0,Y 295.601,Z 1034.086,A -85,B 0,C 180,E1 3061.357,E2 3061.357} C_VEL
LIN {X 0,Y 304.981,Z 1013.562,A -85,B 0,C 180,E1 3060.737,E2 3060.737} C_VEL
LIN {X 0,Y 313.207,Z 991.54,A -85,B 0,C 180,E1 3060.216,E2 3060.216} C_VEL
LIN {X 0,Y 319.956,Z 969.149,A -85,B 0,C 180,E1 3059.795,E2 3059.795} C_VEL
LIN {X 0,Y 325.06,Z 945.918,A -85,B 0,C 180,E1 3059.463,E2 3059.463} C_VEL
LIN {X 0,Y 329.164,Z 918.105,A -85,B 0,C 180,E1 3059.132,E2 3059.132} C_VEL
LIN {X 0,Y 339.777,Z 830.39,A -85,B 0,C 180,E1 3058.103,E2 3058.103} C_VEL
LIN {X 0,Y 339.633,Z 831.455,A -85,B 0,C 180,E1 3055.948,E2 3055.948} C_VEL
LIN {X 0,Y 339.606,Z 831.832,A -85,B 0,C 180,E1 3055.786,E2 3055.786} C_VEL
LIN {X 0,Y 326.428,Z 938.715,A -85,B 0,C 180,E1 3054.608,E2 3054.608} C_VEL
LIN {X 0,Y 321.75,Z 962.302,A -85,B 0,C 180,E1 3054.324,E2 3054.324} C_VEL
LIN {X 0,Y 315.668,Z 984.936,A -85,B 0,C 180,E1 3054.028,E2 3054.028} C_VEL
LIN {X 0,Y 308.169,Z 1006.3,A -85,B 0,C 180,E1 3053.666,E2 3053.666} C_VEL
LIN {X 0,Y 299.075,Z 1027.782,A -85,B 0,C 180,E1 3053.176,E2 3053.176} C_VEL
LIN {X 0,Y 288.882,Z 1047.768,A -85,B 0,C 180,E1 3052.573,E2 3052.573} C_VEL
LIN {X 0,Y 275.838,Z 1069.523,A -85,B 0,C 180,E1 3051.717,E2 3051.717} C_VEL
LIN {X 0,Y 263.356,Z 1087.48,A -85,B 0,C 180,E1 3050.793,E2 3050.793} C_VEL
LIN {X 0,Y 248.817,Z 1105.607,A -85,B 0,C 180,E1 3049.581,E2 3049.581} C_VEL
LIN {X 0,Y 233.948,Z 1121.984,A -85,B 0,C 180,E1 3048.156,E2 3048.156} C_VEL
LIN {X 0,Y 217.169,Z 1138.027,A -85,B 0,C 180,E1 3046.277,E2 3046.277} C_VEL
LIN {X 0,Y 199.771,Z 1152.722,A -85,B 0,C 180,E1 3043.938,E2 3043.938} C_VEL
LIN {X 0,Y 182.777,Z 1165.301,A -85,B 0,C 180,E1 3041.151,E2 3041.151} C_VEL
LIN {X 0,Y 164.617,Z 1177.148,A -85,B 0,C 180,E1 3037.402,E2 3037.402} C_VEL
LIN {X 0,Y 147.326,Z 1187.116,A -85,B 0,C 180,E1 3032.755,E2 3032.755} C_VEL
LIN {X 0,Y 130.499,Z 1195.591,A -85,B 0,C 180,E1 3026.63,E2 3026.63} C_VEL
LIN {X 0,Y 114.892,Z 1202.687,A -85,B 0,C 180,E1 3018.454,E2 3018.454} C_VEL
LIN {X 0,Y 102.604,Z 1207.706,A -85,B 0,C 180,E1 3008.585,E2 3008.585} C_VEL
LIN {X 0,Y 92.884,Z 1211.58,A -85,B 0,C 180,E1 2994.823,E2 2994.823} C_VEL
LIN {X 0,Y 88.954,Z 1213.301,A -85,B 0,C 180,E1 2982.331,E2 2982.331} C_VEL
LIN {X 0,Y 88.082,Z 1213.875,A -85,B 0,C 180,E1 2970.65,E2 2970.65} C_VEL
LIN {X 0,Y 88.74,Z 1213.461,A -85,B 0,C 180,E1 2958.957,E2 2958.957} C_VEL
LIN {X 0,Y 92.574,Z 1211.74,A -85,B 0,C 180,E1 2945.769,E2 2945.769} C_VEL
LIN {X 0,Y 101.126,Z 1208.398,A -85,B 0,C 180,E1 2932.906,E2 2932.906} C_VEL
LIN {X 0,Y 112.975,Z 1203.542,A -85,B 0,C 180,E1 2922.729,E2 2922.729} C_VEL
LIN {X 0,Y 129.133,Z 1196.357,A -85,B 0,C 180,E1 2913.884,E2 2913.884} C_VEL
LIN {X 0,Y 145.658,Z 1188.158,A -85,B 0,C 180,E1 2907.686,E2 2907.686} C_VEL
LIN {X 0,Y 162.852,Z 1178.37,A -85,B 0,C 180,E1 2902.935,E2 2902.935} C_VEL
LIN {X 0,Y 180.069,Z 1167.446,A -85,B 0,C 180,E1 2899.275,E2 2899.275} C_VEL
LIN {X 0,Y 196.986,Z 1155.09,A -85,B 0,C 180,E1 2896.399,E2 2896.399} C_VEL
LIN {X 0,Y 214.334,Z 1140.89,A -85,B 0,C 180,E1 2893.997,E2 2893.997} C_VEL
LIN {X 0,Y 230.133,Z 1126.084,A -85,B 0,C 180,E1 2892.163,E2 2892.163} C_VEL
LIN {X 0,Y 247.146,Z 1107.941,A -85,B 0,C 180,E1 2890.49,E2 2890.49} C_VEL
LIN {X 0,Y 261.387,Z 1090.576,A -85,B 0,C 180,E1 2889.284,E2 2889.284} C_VEL
LIN {X 0,Y 274.823,Z 1071.6,A -85,B 0,C 180,E1 2888.277,E2 2888.277} C_VEL
LIN {X 0,Y 286.897,Z 1052.092,A -85,B 0,C 180,E1 2887.475,E2 2887.475} C_VEL
LIN {X 0,Y 297.591,Z 1031.563,A -85,B 0,C 180,E1 2886.828,E2 2886.828} C_VEL
LIN {X 0,Y 307.313,Z 1009.489,A -85,B 0,C 180,E1 2886.302,E2 2886.302} C_VEL
LIN {X 0,Y 314.646,Z 989.103,A -85,B 0,C 180,E1 2885.943,E2 2885.943} C_VEL
LIN {X 0,Y 321.588,Z 964.544,A -85,B 0,C 180,E1 2885.61,E2 2885.61} C_VEL
LIN {X 0,Y 326.425,Z 941.205,A -85,B 0,C 180,E1 2885.327,E2 2885.327} C_VEL
LIN {X 0,Y 332.913,Z 890.265,A -85,B 0,C 180,E1 2884.761,E2 2884.761} C_VEL
LIN {X 0,Y 339.971,Z 831.92,A -85,B 0,C 180,E1 2884.091,E2 2884.091} C_VEL
LIN {X 0,Y 340.049,Z 830.959,A -85,B 0,C 180,E1 2882.528,E2 2882.528} C_VEL
LIN {X 0,Y 340.103,Z 831,A -85,B 0,C 180,E1 2881.874,E2 2881.874} C_VEL
LIN {X 0,Y 326.911,Z 937.547,A -85,B 0,C 180,E1 2880.642,E2 2880.642} C_VEL
LIN {X 0,Y 322.209,Z 961.228,A -85,B 0,C 180,E1 2880.327,E2 2880.327} C_VEL
LIN {X 0,Y 316.229,Z 983.542,A -85,B 0,C 180,E1 2879.956,E2 2879.956} C_VEL
LIN {X 0,Y 308.468,Z 1005.665,A -85,B 0,C 180,E1 2879.477,E2 2879.477} C_VEL
LIN {X 0,Y 298.942,Z 1027.978,A -85,B 0,C 180,E1 2878.85,E2 2878.85} C_VEL
LIN {X 0,Y 289.105,Z 1047.2,A -85,B 0,C 180,E1 2878.171,E2 2878.171} C_VEL
LIN {X 0,Y 275.999,Z 1069.049,A -85,B 0,C 180,E1 2877.204,E2 2877.204} C_VEL
LIN {X 0,Y 263.054,Z 1087.649,A -85,B 0,C 180,E1 2876.156,E2 2876.156} C_VEL
LIN {X 0,Y 248.47,Z 1105.794,A -85,B 0,C 180,E1 2874.844,E2 2874.844} C_VEL
LIN {X 0,Y 232.596,Z 1123.243,A -85,B 0,C 180,E1 2873.214,E2 2873.214} C_VEL
LIN {X 0,Y 216.459,Z 1138.681,A -85,B 0,C 180,E1 2871.301,E2 2871.301} C_VEL
LIN {X 0,Y 203.719,Z 1149.718,A -85,B 0,C 180,E1 2869.551,E2 2869.551} C_VEL
LIN {X 0,Y 197.825,Z 1154.381,A -85,B 0,C 180,E1 2868.982,E2 2868.982} C_VEL
LIN {X 0,Y 181.279,Z 1165.648,A -85,B 0,C 180,E1 2868.328,E2 2868.328} C_VEL
LIN {X 0,Y 175.041,Z 1169.634,A -85,B 0,C 180,E1 2867.581,E2 2867.581} C_VEL
LIN {X 0,Y 157.164,Z 1180.825,A -85,B 0,C 180,E1 2863.872,E2 2863.872} C_VEL
LIN {X 0,Y 137.574,Z 1191.684,A -85,B 0,C 180,E1 2858.478,E2 2858.478} C_VEL
LIN {X 0,Y 121.012,Z 1199.818,A -85,B 0,C 180,E1 2852.139,E2 2852.139} C_VEL
LIN {X 0,Y 104.937,Z 1206.891,A -85,B 0,C 180,E1 2843.109,E2 2843.109} C_VEL
LIN {X 0,Y 92.573,Z 1212.038,A -85,B 0,C 180,E1 2832.04,E2 2832.04} C_VEL
LIN {X 0,Y 83.825,Z 1215.672,A -85,B 0,C 180,E1 2817.722,E2 2817.722} C_VEL
LIN {X 0,Y 80.415,Z 1217.503,A -85,B 0,C 180,E1 2804.1,E2 2804.1} C_VEL
LIN {X 0,Y 80.009,Z 1218.107,A -85,B 0,C 180,E1 2792.865,E2 2792.865} C_VEL
LIN {X 0,Y 79.995,Z 1218.05,A -85,B 0,C 180,E1 2785.699,E2 2785.699} C_VEL
LIN {X 0,Y 80.538,Z 1217.377,A -85,B 0,C 180,E1 2774.888,E2 2774.888} C_VEL
LIN {X 0,Y 84.1,Z 1215.514,A -85,B 0,C 180,E1 2761.605,E2 2761.605} C_VEL
LIN {X 0,Y 93.549,Z 1211.541,A -85,B 0,C 180,E1 2746.84,E2 2746.84} C_VEL
LIN {X 0,Y 105.611,Z 1206.526,A -85,B 0,C 180,E1 2736.416,E2 2736.416} C_VEL
LIN {X 0,Y 122.515,Z 1198.97,A -85,B 0,C 180,E1 2727.182,E2 2727.182} C_VEL
LIN {X 0,Y 139.219,Z 1190.714,A -85,B 0,C 180,E1 2720.99,E2 2720.99} C_VEL
LIN {X 0,Y 157.157,Z 1180.651,A -85,B 0,C 180,E1 2716.12,E2 2716.12} C_VEL
LIN {X 0,Y 175.063,Z 1169.422,A -85,B 0,C 180,E1 2712.405,E2 2712.405} C_VEL
LIN {X 0,Y 193.554,Z 1156.113,A -85,B 0,C 180,E1 2709.368,E2 2709.368} C_VEL
LIN {X 0,Y 211.534,Z 1141.534,A -85,B 0,C 180,E1 2706.973,E2 2706.973} C_VEL
LIN {X 0,Y 227.885,Z 1126.375,A -85,B 0,C 180,E1 2705.143,E2 2705.143} C_VEL
LIN {X 0,Y 244.918,Z 1108.433,A -85,B 0,C 180,E1 2703.511,E2 2703.511} C_VEL
LIN {X 0,Y 259.174,Z 1091.278,A -85,B 0,C 180,E1 2702.317,E2 2702.317} C_VEL
LIN {X 0,Y 273.232,Z 1071.779,A -85,B 0,C 180,E1 2701.258,E2 2701.258} C_VEL
LIN {X 0,Y 285.516,Z 1052.225,A -85,B 0,C 180,E1 2700.421,E2 2700.421} C_VEL
LIN {X 0,Y 296.572,Z 1031.295,A -85,B 0,C 180,E1 2699.71,E2 2699.71} C_VEL
LIN {X 0,Y 306.492,Z 1009.035,A -85,B 0,C 180,E1 2699.113,E2 2699.113} C_VEL
LIN {X 0,Y 314.038,Z 988.239,A -85,B 0,C 180,E1 2698.682,E2 2698.682} C_VEL
LIN {X 0,Y 320.909,Z 964.174,A -85,B 0,C 180,E1 2698.291,E2 2698.291} C_VEL
LIN {X 0,Y 325.619,Z 941.864,A -85,B 0,C 180,E1 2698.004,E2 2698.004} C_VEL
LIN {X 0,Y 330.476,Z 905.747,A -85,B 0,C 180,E1 2697.599,E2 2697.599} C_VEL
LIN {X 0,Y 337.457,Z 848.699,A -85,B 0,C 180,E1 2696.962,E2 2696.962} C_VEL
LIN {X 0,Y 326.164,Z 938.822,A -85,B 0,C 180,E1 2696.014,E2 2696.014} C_VEL
LIN {X 0,Y 321.4,Z 962.432,A -85,B 0,C 180,E1 2695.749,E2 2695.749} C_VEL
LIN {X 0,Y 315.186,Z 985.227,A -85,B 0,C 180,E1 2695.478,E2 2695.478} C_VEL
LIN {X 0,Y 307.631,Z 1006.543,A -85,B 0,C 180,E1 2695.152,E2 2695.152} C_VEL
LIN {X 0,Y 298.233,Z 1028.422,A -85,B 0,C 180,E1 2694.698,E2 2694.698} C_VEL
LIN {X 0,Y 288.448,Z 1047.435,A -85,B 0,C 180,E1 2694.176,E2 2694.176} C_VEL
LIN {X 0,Y 275.773,Z 1068.51,A -85,B 0,C 180,E1 2693.427,E2 2693.427} C_VEL
LIN {X 0,Y 263.16,Z 1086.559,A -85,B 0,C 180,E1 2692.59,E2 2692.59} C_VEL
LIN {X 0,Y 248.212,Z 1105.119,A -85,B 0,C 180,E1 2691.467,E2 2691.467} C_VEL
LIN {X 0,Y 232.906,Z 1121.799,A -85,B 0,C 180,E1 2690.142,E2 2690.142} C_VEL
LIN {X 0,Y 216.34,Z 1137.464,A -85,B 0,C 180,E1 2688.464,E2 2688.464} C_VEL
LIN {X 0,Y 199.54,Z 1151.582,A -85,B 0,C 180,E1 2686.433,E2 2686.433} C_VEL
LIN {X 0,Y 182.133,Z 1164.291,A -85,B 0,C 180,E1 2683.883,E2 2683.883} C_VEL
LIN {X 0,Y 163.423,Z 1176.355,A -85,B 0,C 180,E1 2680.425,E2 2680.425} C_VEL
LIN {X 0,Y 146.288,Z 1185.988,A -85,B 0,C 180,E1 2676.329,E2 2676.329} C_VEL
LIN {X 0,Y 127.753,Z 1195.114,A -85,B 0,C 180,E1 2670.313,E2 2670.313} C_VEL
LIN {X 0,Y 111.699,Z 1202.089,A -85,B 0,C 180,E1 2662.813,E2 2662.813} C_VEL
LIN {X 0,Y 97.474,Z 1207.516,A -85,B 0,C 180,E1 2652.61,E2 2652.61} C_VEL
LIN {X 0,Y 86.977,Z 1211.351,A -85,B 0,C 180,E1 2639.624,E2 2639.624} C_VEL
LIN {X 0,Y 81.396,Z 1213.378,A -85,B 0,C 180,E1 2624.949,E2 2624.949} C_VEL
LIN {X 0,Y 80.096,Z 1214.036,A -85,B 0,C 180,E1 2612.146,E2 2612.146} C_VEL
LIN {X 0,Y 80.495,Z 1213.836,A -85,B 0,C 180,E1 2600.707,E2 2600.707} C_VEL
LIN {X 0,Y 84.377,Z 1212.273,A -85,B 0,C 180,E1 2585.497,E2 2585.497} C_VEL
LIN {X 0,Y 92.808,Z 1209.309,A -85,B 0,C 180,E1 2572.115,E2 2572.115} C_VEL
